// TwinCAT 3 PLC project PLC_HMI_ACCT_1
// ProgramVersion: 3.1.4026.19
// libraries:
//   Tc2_DataExchange, * (Beckhoff Automation GmbH)
//   Tc2_IoFunctions, * (Beckhoff Automation GmbH)
//   Tc2_MC2, * (Beckhoff Automation GmbH)
//   Tc2_Standard, * (Beckhoff Automation GmbH)
//   Tc2_System, * (Beckhoff Automation GmbH)
//   Tc2_Utilities, * (Beckhoff Automation GmbH)
//   Tc3_Database, * (Beckhoff Automation GmbH)
//   Tc3_EventLogger, * (Beckhoff Automation GmbH)
//   Tc3_Module, * (Beckhoff Automation GmbH)
// project tree:
//   DUTs/ ST_Alarm.TcDUT, ST_Error_Station_Handling.TcDUT, ST_Error_Description_Handling.TcDUT, ST_For_Screen.TcDUT, ST_For_Screen_New.TcDUT, ST_Recipe_Changes.TcDUT, ST_UserManagment.TcDUT, S_Information.TcDUT, S_Information_Text.TcDUT, S_LogData.TcDUT
//   FB/ FB_GetSystemTime.TcPOU, FB_Persistent.TcPOU, FB_ReadWriteLogCSV.TcPOU, FB_Save.TcPOU, FB_SaveLineToFile.TcPOU, FB_SaveTextToFile.TcPOU
//   FB/RecipeCSV/ FB_ListSaveCSV.TcPOU, FB_LoadCSV.TcPOU, FB_RecipeSaveCSV.TcPOU, FB_RecipeVariablesSaveCSV.TcPOU
//   FB/RecipeList/ E_FileOpSteps.TcDUT, FB_Load.TcPOU
//   GVLs/ GVL_CFG.TcGVL, GVL_Error.TcGVL, GVL_Gauge.TcGVL, GVL_Recipe.TcGVL, GVL_Screw.TcGVL, GVL_USER.TcGVL
//   NotUsedPOU/ P_50_screw.TcPOU, P_Error_Handling.TcPOU
//   / PlcTask.TcTTO
//   POUs/ADS/ P_ADS_Gauge.TcPOU, P_ADS_OEE.TcPOU, P_ADS_Screw.TcPOU
//   POUs/DataLogging/ p_24h_C1_2.TcPOU, p_24h_C2_2.TcPOU, P_ArrayToFile.TcPOU, P_CameraFlip.TcPOU, P_Gauge_Measures.TcPOU, P_OEE_Raport.TcPOU, P_Recipebackup.TcPOU, P_RecipeChange.TcPOU, P_ScrewersCharts_1.TcPOU, P_ScrewersCharts_2.TcPOU
//   POUs/ MAIN.TcPOU, P_Time.TcPOU
//   POUs/Persistent/ P_Persistent.TcPOU, P_PersistentDataSave.TcPOU
//   POUs/Users/ P_UserManagment.TcPOU
// (motion and I/O tree: see PLC project programplc)
// real-time tasks:
//   TASK MainTask: cycle T#3ms, priority 20, ADS port 350
//   TASK SafetyTask: cycle T#10ms, priority 22, ADS port 351
//   TASK WeightTask: cycle T#2ms, priority 19, ADS port 354
//   TASK PlcTask: cycle T#10ms, priority 21, ADS port 355
//   TASK TaskToRefreshEAP: cycle T#1ms, priority 12, ADS port 301
// variable links:

CONFIGURATION PLC_HMI_ACCT_1
    RESOURCE PLC ON TwinCAT3
        TASK PlcTask(INTERVAL := T#10ms, PRIORITY := 21);
        PROGRAM MAIN WITH PlcTask : MAIN;
    END_RESOURCE
END_CONFIGURATION

// ---- DUTs/ST_Alarm.TcDUT
TYPE ST_Alarm :
STRUCT
	sTekst1				: WSTRING(255);
	sTekst2				: WSTRING(255);
	sTekst3				: WSTRING(255);
	dtUtworzenia		: DT;
	iNumer				: INT;
	historical_alarm	: WSTRING(1000);
END_STRUCT
END_TYPE

// ---- DUTs/ST_Error_Station_Handling.TcDUT
TYPE ST_Error_Station_Handling :
STRUCT
	udiStationInError			:UDINT;
	wsStasionInError				:WSTRING(255);
END_STRUCT
END_TYPE

// ---- DUTs/ST_Error_Description_Handling.TcDUT
TYPE ST_Error_Description_Handling :
STRUCT
	udiStationErrorCode		:UDINT;
	wsStationErrorDescription	:WSTRING(255);	
END_STRUCT
END_TYPE

// ---- DUTs/ST_For_Screen.TcDUT
TYPE ST_For_Screen :
STRUCT
	data				:WSTRING(255);
	alarmy				:WSTRING(1000);
	user				:WSTRING(80);
	bErrorOccure		:BOOL := FALSE;
END_STRUCT
END_TYPE

// ---- DUTs/ST_For_Screen_New.TcDUT
TYPE ST_For_Screen_New :
STRUCT
	data				:WSTRING(255);
	alarmy				:WSTRING(1000);
	alarmy_id			:UDINT;
	stacja				:UDINT;
	user				:WSTRING(80);
	bErrorOccure		:BOOL := FALSE;
END_STRUCT
END_TYPE

// ---- DUTs/ST_Recipe_Changes.TcDUT
TYPE ST_Recipe_Changes :
STRUCT
	old_value :LREAL;
	new_value :LREAL;
	who_changed :WSTRING(200);
	when_changed :DT;	
	which_param_name :WSTRING(200);
	which_param_var	 :WSTRING(200);	
	which_param_cntr :WSTRING(200);
	which_recipe :WSTRING(200);
	
END_STRUCT
END_TYPE

// ---- DUTs/ST_UserManagment.TcDUT
TYPE ST_UserManagment :
STRUCT
	userID 				:	INT;			//numer porządkowy użytkownika
//	domain				:	STRING(80);
	enabled				:	BOOL;
	userLogin			:	STRING(80);		//login do zalogowania
	userNameSurname 	:	WSTRING(255);	//imię i nazwisko
	userNameSurnameNumber	:UINT;
	password			:	STRING(255);	//hasło kalwiaturowe
	passwordRFID		:	STRING(255);	//hasło rfid
	passwordQR			:	STRING(255);	//hasło qr
	userGroup			:	STRING(80);		//grupa użytkowników
	userGropuNumber		:	UINT;			//numer grupy
//	autoLogOff			:	STRING(80);		//czas do wylogowania
//	locale				:	STRING(80);		//gdzie zapisujemy
//	timeFormatlocale	:	STRING(80);		//format godziny
//	timeZone			:	STRING(80);		//strefa czasowa
	signedPassword		:	STRING(80);		//hasło przekazywane do HMI
END_STRUCT
END_TYPE

// ---- DUTs/S_Information.TcDUT
(*
Nazwa:			S_Error
Opis:			Struktura bledu
Wersja:			v0.2
Data:			2018-10-10
Autor:			TW
Urzadzenia:		
Konfiguracja:	
Info:
- dodano string2
*)
TYPE S_Information :
STRUCT 
	udiID				: UDINT;
	wsDescription		: WSTRING;
END_STRUCT
END_TYPE

// ---- DUTs/S_Information_Text.TcDUT
(*
Nazwa:			S_Error
Opis:			Struktura bledu
Wersja:			v0.2
Data:			2018-10-10
Autor:			TW
Urzadzenia:		
Konfiguracja:	
Info:
- dodano string2
*)
TYPE S_Information_Text :
STRUCT 
	desc				: WSTRING;
	wsDescription		: WSTRING;
END_STRUCT
END_TYPE

// ---- DUTs/S_LogData.TcDUT
TYPE S_LogData :
STRUCT
END_STRUCT
END_TYPE

// ---- FB/RecipeList/E_FileOpSteps.TcDUT
{attribute 'qualified_only'}
{attribute 'strict'}
TYPE E_FileOpSteps :
(
	eNop 					:=	0,
	eStartOpen				:=	10,
	eWaitOpen				:=	20,
	eStartOper				:=	30,
	eWaitOper				:=	40,
	eStartClose				:=	50,
	eWaitClose				:=	60
);
END_TYPE

// ---- GVLs/GVL_CFG.TcGVL
{attribute 'qualified_only'}
VAR_GLOBAL PERSISTENT
	//butelki
	bBottleBuPu :BOOL:=FALSE;
	bBottlePI :BOOL:=TRUE;
	bBottleUBF :BOOL:=TRUE;
	bNoBottleFeed	:BOOL:=FALSE;
	
	//nasadki
	bCapUCF :BOOL:=TRUE;
	bCapSO :BOOL:=FALSE;
	bCapWibro :BOOL:=FALSE;
	bCapGiraffe :BOOL:=FALSE;
	bNoCapFeed	:BOOL:=FALSE;
	
	//maszyna
	bPlatinsCFG :BOOL:=TRUE;
	bTwoPhaseCFG :BOOL:=TRUE;;
	bAirless :BOOL:=FALSE;
	bROPP :BOOL:=FALSE;;
	
	sIP	:STRING:='192.168.40.180.1.1';
	sPort :T_AmsPort:=851;
	
	sRightTime	:STRING;
	tbreakTime_1:STRING:='10:35:00';
	tbreakTime_2:STRING:='14:35:00';
	bBreakReset:BOOL;
	
	bWenglorCapPutted :BOOL;
	bWenglorCapCorrect :BOOL;
	
END_VAR

// ---- GVLs/GVL_Error.TcGVL
{attribute 'qualified_only'}
(**VAR_GLOBAL PERSISTENT
	udi_Station_In_Error			:UDINT;
	udi_Station_In_Error_Code		:UDINT;
	ws_Stasion_In_Error				:WSTRING;
	ws_Station_Error_Description		:WSTRING(255);
	ws_Station_Error_Description_2	:WSTRING(255);
	A_Error_station	:ARRAY[0..100] OF ST_Error_Station_Handling; 
	A_Error_description	:ARRAY[0..500] OF ST_Error_Description_Handling;
	
	b_empy_error					:BOOL;
	b_new_system					:BOOL;
	
	sVisGuid						:STRING;
	
	b_reset_event_logger :BOOL;
END_VAR**)
VAR_GLOBAL
	b_reset_event_logger :BOOL;
	logowanie_krok: INT;
	b_cameras_ivms:BOOL;
END_VAR

// ---- GVLs/GVL_Gauge.TcGVL
{attribute 'qualified_only'}
VAR_GLOBAL
	//input
	lr_WeightMass_recipe	:LREAL;
	lr_Dispencer1WeightMeasured	:LREAL;
	lr_Dispencer2WeightMeasured	:LREAL;
	lr_Dispencer3WeightMeasured	:LREAL;
	lr_Dispencer4WeightMeasured	:LREAL;
	lr_Tolerance_Low			:LREAL;
	lr_Tolerance_High			:LREAL;
	lr_weight_measured_1		:LREAL;
	lr_weight_measured_2		:LREAL;
	lr_weight_measured_3		:LREAL;
	lr_weight_measured_4		:LREAL;
	
	lr_mass_value_1				:LREAL;
	lr_mass_value_2				:LREAL;
	lr_mass_value_3				:LREAL;
	lr_mass_value_4				:LREAL;
	
	
	//output
	lr_out_max_weight_value :LREAL;
	lr_out_min_tolerance_low :LREAL;
	lr_out_max_tolerance_high :LREAL;
	
	lr_out_weight_measured_1 :LREAL;
	lr_out_weight_measured_2 :LREAL;
	lr_out_weight_measured_3 :LREAL;
	lr_out_weight_measured_4 :LREAL;
	
	s_actual_weight_1	:STRING;
	s_actual_weight_2	:STRING;	
	s_actual_weight_3	:STRING;
	s_actual_weight_4	:STRING;
	
	s_actual_weight_1_diff	:STRING;
	s_actual_weight_2_diff	:STRING;
	s_actual_weight_3_diff	:STRING;
	s_actual_weight_4_diff	:STRING;

	s_actual_corr_1		:STRING;
	s_actual_corr_2		:STRING;
	s_actual_corr_3		:STRING;
	s_actual_corr_4		:STRING;	
	
	s_actual_dose_1		:STRING;
	s_actual_dose_2		:STRING;
	s_actual_dose_3		:STRING;
	s_actual_dose_4		:STRING;
	
	lr_corr_add_1	:LREAL;
	lr_corr_sub_1	:LREAL;
	lr_corr_add_2	:LREAL;
	lr_corr_sub_2	:LREAL;
	lr_corr_add_3	:LREAL;
	lr_corr_sub_3	:LREAL;
	lr_corr_add_4	:LREAL;
	lr_corr_sub_4	:LREAL;
	
	s_actual_torque_1	:STRING;
	s_actual_torque_2	:STRING;
	s_actual_torque_diff_1		:STRING;
	s_actual_torque_diff_2		:STRING;
	
	s_actual_level_1	:STRING;
	s_actual_level_2	:STRING;
	
	lr_out_torque_low_1		:LREAL;
	lr_out_torque_low_2		:LREAL;
	lr_out_torque_high_1		:LREAL;
	lr_out_torque_high_2		:LREAL;	
	
	s_out_weight_measured_1 :STRING;
	s_out_weight_measured_2 :STRING;
	s_out_weight_measured_3 :STRING;
	s_out_weight_measured_4 :STRING;

	lr_diff_dispencer_1:LREAL;
	lr_diff_dispencer_2:LREAL;
	
	s_time_mainscreen:WSTRING(80);
	
	bDosingTwoPhasesShow	:BOOL;
END_VAR

// ---- GVLs/GVL_Recipe.TcGVL
{attribute 'qualified_only'}
VAR_GLOBAL PERSISTENT
	b_recipe_backup	:BOOL;
	
	b_recipe_bool_change :BOOL; //sygnał, że ktoś zmienił parametr bool
	b_recipe_real_change :BOOL; //sygnał, że ktoś zmienił parametr inny
	i_recipe_change :INT;
	lr_recipe_change :LREAL; //stara wartość w polu lr_param
	
	b_recipe_change_1 :BOOL;
	i_recipe_change_1 :INT;
	lr_recipe_change_1 :LREAL; //nowa wartość w polu lr_param
	
	s_recipe_change    :WSTRING(200); //kto zmienił parametr
	s_recipe_change_1  :WSTRING(200); //jaki parametr
	s_recipe_change_2  :WSTRING(200); //zmienna receptury
	s_recipe_change_3  :WSTRING(300); //zmienna do kontrolki
	b_old_recipe_param :BOOL; //stara wartość parametru b_param
	b_new_recipe_param :BOOL; //nowa wartość parametru b_param
	

	
	s_recipe_value :STRING;
	ArRecipeChanges: ARRAY [0..500] OF st_recipe_changes;	
	s_recipe_name :WSTRING(200); //nazwa receptury
	s_recupe_change_4 :WSTRING(200);
	b_recipe_changes_clear :BOOL:=FALSE;
END_VAR

// ---- GVLs/GVL_Screw.TcGVL
{attribute 'qualified_only'}
VAR_GLOBAL
	 aLast50Screw1: ARRAY[1..501] OF LREAL;
	 aLast50Screw2: ARRAY[1..501] OF LREAL;
	 bExport:BOOL;
	 a50ScrewSetted1: ARRAY[1..501] OF LREAL;
	 a50ScrewSetted2: ARRAY[1..501] OF LREAL;
END_VAR

// ---- GVLs/GVL_USER.TcGVL
{attribute 'qualified_only'}
VAR_GLOBAL PERSISTENT
	user_array 					: ARRAY[1..100] OF ST_UserManagment;  // Tablica użytkowników
    currentUser 				: INT := 1;  // Indeks bieżącego użytkownika (zaczyna od 1)
	outside_login_pool			:STRING(255);  
	currentUserName 			:WSTRING(255);
	currentUserGroup			:STRING(80);
	currentUserGroupNumber		:UINT;
	putted_user_password		:STRING(255);  //pole w które użytkownik wpisuje hasło
	newuserNameSurname 			:WSTRING(255);	//imię i nazwisko
	newpassword					:STRING(255);	//hasło
	newpasswordRFID				:STRING(255);	//hasło rfid
	newpasswordQR				:STRING(255);	//hasło qr
	newuserGroup				:STRING(80);		//grupa użytkowników
	newuserGroupNumber			:UINT;
	newautoLogOff				:STRING(80);			//czas do wylogowania
	actual_editted_user			:WSTRING(255);	//wybór aktualnie edytowanego użytkownika
	edituserNameSurname 		:WSTRING(255);	//imię i nazwisko
	editpassword				:STRING(255);	//hasło
	editpasswordRFID			:STRING(255);	//hasło rfid
	editpasswordQR				:STRING(255);	//hasło qr
	edituserGroup				:STRING(80);	//grupa użytkowników
	editUserGroupNumber			:UINT;
	editautoLogOff				:STRING(80);	//czas do wylogowania


END_VAR
VAR_GLOBAL
	new_user_add_error			:BOOL;
	edit_user_error				:BOOL;
	bwait						:BOOL;
	delete_user					:BOOL;
	delete_user_accept			:BOOL;
	delete_user_error			:BOOL;
	choosen_to_delete			:WSTRING(255);
	user_deleted_succes			:BOOL;
	password_to_log_in			:STRING(80); //hasło do pola (1 z 5 (adm, opr, ser, tech, mech	
	b_rewrite_users_after_issues:BOOL:=FALSE;
	b_user_drop_the_login		:BOOL;
	i_choosen_language 			:INT:=1;
	outside_accept_login		:BOOL;
	logout						:BOOL;
	user_try_to_log				:BOOL;
	user_accept_to_log_in		:BOOL;
	no_user_found				:BOOL;
	user_succesed_log			:BOOL;
	edit_user_qr_or_rfid_password :BOOL;		//edycja kodów rfid lub qr
	new_user_added				:BOOL;		//dodano użytkownika w PLC
	user_eddited				:BOOL; 		//zedytowano użytkownika w PLC
	b_new_users					:BOOL;		//wgranie uzytkowników
	new_user					:BOOL;			//inicjalizacja dodawania nowego użytkownika
	new_user_accept				:BOOL;			//akceptacja dodania nowego użytkownika
	edit_user					:BOOL;				//inicjalizacja edycji użytkownika
	edit_user_accept			:BOOL;			//akceptacja edycji użytkownika
	actualUserOn_UserName		:STRING(80);
	b_rewrite_main_users		:BOOL:=FALSE;
	string_of_properties 		: STRING(1000);  // String z HMI z danymi użytkowników
END_VAR

// ---- POUs/MAIN.TcPOU
PROGRAM MAIN
VAR
		
END_VAR

//P_ADS_1();
P_Time();
//P_History_New();
P_UserManagment();
P_Recipebackup();
P_Gauge_Measures();
P_ADS_Gauge();
//P_ADS_Err();
//P_Error_Handling();
P_RecipeChange();
P_ArrayToFile();
P_ScrewersCharts_1();
P_ScrewersCharts_2();
P_ADS_Screw();
P_24h_C1_2();
P_24h_C2_2();
//P_HistoryWarning();
P_CameraFlip();
//P_EventLogger();
//P030_Recipes();
//P010_AlarmsWarningsInfosLogs();
//P020_RtcEffectivityOEE();
//P009_ReadSavePersistent();
P_OEE_Raport();
P_ADS_OEE();
P_PersistentDataSave();
P_Persistent();

END_PROGRAM

// ---- POUs/P_Time.TcPOU
PROGRAM P_Time
VAR
    fbSystemTime : GETSYSTEMTIME;
	fbSystemTime2 : FB_GetSystemTime;
    timeAsFileTime : T_FILETIME;
    timeAsDT : DT;
	actual_date_meawhile :DT;
	s_time_mainscreen	:WSTRING(80);
	tonBreakTurnOff 	:TON;
END_VAR

tonBreakTurnOff(IN:=gvl_cfg.bBreakReset,PT:=T#5S);
fbSystemTime2(bEnable:=TRUE);
fbSystemTime(
    timeLoDW => timeAsFileTime.dwLowDateTime,
    timeHiDW => timeAsFileTime.dwHighDateTime 
);
(*timeAsDT := FILETIME_TO_DT(timeAsFileTime);
actual_date_meawhile:=timeAsDT;
actual_date_meawhile := actual_date_meawhile + T#2H;
s_time_mainscreen := DT_TO_WSTRING(actual_date_meawhile);
s_time_mainscreen := WRIGHT(s_time_mainscreen, WLEN(s_time_mainscreen) - 3);
gvl_his.s_time_mainscreen:=s_time_mainscreen;
gvl_cfg.wsRightTime:=WRIGHT(s_time_mainscreen,8);*)
timeAsDT :=fbSystemTime2.dtActTime;
actual_date_meawhile:=timeAsDT;
s_time_mainscreen := DT_TO_WSTRING(actual_date_meawhile);
s_time_mainscreen := WRIGHT(s_time_mainscreen, WLEN(s_time_mainscreen) - 3 );
gvl_gauge.s_time_mainscreen:=s_time_mainscreen;


IF gvl_cfg.sRightTime = gvl_cfg.tbreakTime_1 OR gvl_cfg.sRightTime = gvl_cfg.tbreakTime_2 THEN
	gvl_cfg.bBreakReset:=TRUE;
END_IF

IF tonBreakTurnOff.Q THEN
	gvl_cfg.bBreakReset:=FALSE;
END_IF

END_PROGRAM

// ---- FB/FB_GetSystemTime.TcPOU
(****************************************************************************************)
(*							Beckhoff Automation Poland									*)
(*								FB_GetSystemTime  v1.2									*)
(*									26.07.2013											*)
(*		v1.2 - zmiana nazwy bloku z FB_Time na FB_GetSystemTime, dodanie wyjscia DT		*)
(*		v1.1 - dodano na wyjściu zmienną czasu w formie struktury TIMESTRUCT 			*)
(*				Blok funkcyjny podający dokładną datę w odrębnych zmiennych				*)
(*						może być wywołany raz w programie PLC							*)
(*						Wymaga dodania biblioteki TcUtilities.lib						*)
(*______________________________________________________________________________________*)
FUNCTION_BLOCK FB_GetSystemTime
VAR_INPUT
	bEnable:			BOOL;				(*Aktywuje pobieranie czasu systemowego*)
END_VAR
VAR_OUTPUT
	stActTime			:	TIMESTRUCT;
	dtActTime: DT;
(*Poszczególne składowe daty*)
	wYear 				:	WORD;
	wMonth 				:	WORD;
	wDayOfWeek 			: 	WORD;
	wDay 				:	WORD;
	wHour 				:	WORD;
	wMinute 			:	WORD;
	wSecond 			:	WORD;
	wMilliseconds 		: 	WORD;
END_VAR
VAR
	fbGetTime			:	NT_GetTime;
	Get					:	TON;
END_VAR
VAR CONSTANT
	tFrequency			:	TIME			:= T#1s;				(*Częstotliwość pobierania czasu*)
END_VAR

Get(IN:= NOT Get.Q AND bEnable, PT:=tFrequency);
fbGetTime(
	NETID:= '',
	START:= Get.Q,
	TMOUT:= T#200ms,
	TIMESTR=>stActTime);

dtActTime 		:= SYSTEMTIME_TO_DT(stActTime);
wDay 			:= stActTime.wDay;
wDayOfWeek 		:= stActTime.wDayOfWeek;
wHour 			:= stActTime.wHour;
wMilliseconds 	:= stActTime.wMilliseconds;
wMinute 		:= stActTime.wMinute;
wMonth 			:= stActTime.wMonth;
wSecond 		:= stActTime.wSecond;
wYear 			:= stActTime.wYear;

END_FUNCTION_BLOCK

// ---- POUs/Users/P_UserManagment.TcPOU
PROGRAM P_UserManagment
VAR	
	user_log				:BOOL 				:= GVL_USER.user_try_to_log;           	//użytkownik wywołał okno logowania
	user_accept				:BOOL 				:= GVL_USER.user_accept_to_log_in;     	//użytkownik zaakceptował hasło
	outside_login_accept	:BOOL				:= gvl_user.outside_accept_login;		//przekazanie potwierdzenia procesu logowania
	user_login_error		:BOOL 				:= GVL_USER.no_user_found;				//brak dopasowanego użytkownika
	user_log_succes			:BOOL 				:= GVL_USER.user_succesed_log;			//zalogowano z powodzeniem
	i,j,z					:INT;														//zmienne dla warunków
	bprzypisanie			:BOOL;
	btest					:BOOL:=FALSE;
	k						:INT;
	userExists				:BOOL;														//zmienne dla programu
	outside_login_pool		:STRING(255)		:= gvl_user.outside_login_pool;												//przekazanie loginu do wizualizacji
	user_password			:STRING(255) 		:= GVL_USER.putted_user_password;		//wprowadzone użytkownikiem hasło
	b_new_users				:BOOL;									
	delayTimer: TON;  // Timer do opóźnienia o 500 ms					//nowe wgranie użytkowników
	allowedGroups : ARRAY[1..5] OF STRING(80) := ['Admin', 'Mechanik', 'Operator', 'Technolog', 'Serwis'];
	allowedGroupsNumber	:ARRAY[1..5] OF UINT:=[1,2,3,4,5];
	validGroup    : BOOL;  // Zmienna do walidacji grupy
    uniqueUser    : BOOL;  // Zmienna sprawdzająca unikalność hasła
    freeSlot      : BOOL;  // Zmienna wskazująca wolne miejsce na nowego użytkownika
	bwait	:BOOL :=gvl_user.bwait; //ekran oczekiwania na plc
	bClear	:BOOL:=FALSE;
	iClearArrayNr :INT;
	
	actual_user : WSTRING(255);
	

	new_user				:BOOL := GVL_USER.new_user;			//inicjalizacja dodania nowego użytkownika
	new_user_accept			:BOOL := GVL_USER.new_user_accept;			//akceptacja dodania użytkownika z ekranu
	new_user_added			:BOOL := GVL_USER.new_user_added;			//udane dodanie użytkownika
	new_user_add_error		:BOOL := GVL_USER.new_user_add_error;			//nieudane dodawanie
	newautoLogOff			:STRING(80) := GVL_USER.newautoLogOff;			//czas do wylogowania
	newuserNameSurname 		:WSTRING(255)  := GVL_USER.newuserNameSurname;	//imię i nazwisko				
	newpassword				:STRING(255) := GVL_USER.newpassword;	//hasło
	newpasswordRFID			:STRING(255) := GVL_USER.newpasswordRFID;	//hasło rfid
	newpasswordQR			:STRING(255) := GVL_USER.newpasswordQR;	//hasło qr
	newuserGroup			:STRING(80) := GVL_USER.newuserGroup;		//grupa użytkowników
	newuserLogoffbetween 	:STRING(80);
	
	edit_user						:BOOL := GVL_USER.edit_user;	//inicjalizacja edycji parametrów użytkownika
	edit_user_accept				:BOOL := GVL_USER.edit_user_accept;	//akceptacja wprowadzonych zmiennych z ekranu
	user_eddited					:BOOL := GVL_USER.user_eddited;	//odpowiedź z plc do hmi - udana edycja
	edit_user_qr_or_rfid_password	:BOOL := GVL_USER.edit_user_qr_or_rfid_password;	//edycja rfid lub qr dopisanego do użytkownika
	edit_user_error					:BOOL := GVL_USER.edit_user_error;			//odpowiedź z plc do hmi - nieudana edycja uzytkownika
	editautoLogOff					:STRING(80) := GVL_USER.editautoLogOff;			//czas do wylogowania użytkownika
	edituserNameSurname 			:WSTRING(255) := GVL_USER.edituserNameSurname ;	//imię i nazwisko
	editpassword					:STRING(255) := GVL_USER.editpassword;	//hasło
	editpasswordRFID				:STRING(255) := GVL_USER.editpasswordRFID;	//hasło rfid
	editpasswordQR					:STRING(255) := GVL_USER.editpasswordQR;	//hasło qr
	edituserGroup					:STRING(80) := GVL_USER.edituserGroup;	//grupa użytkowników
	edituserLogoffbetween 	:STRING(80);

	userExists_2			:BOOL;
	userExists_3			:BOOL;
	
	bFirstCycle				:BOOL := FALSE;
	
	iValueForCheck			:INT;
	logowanie_krok	:INT;
	bLogOffUserReset :BOOL;
	tonLogOffUser :ton;
END_VAR


bFirstCycle:=TRUE; //Symulacja 1 cyklu sterownika
tonLogOffUser(IN:=(NOT (GVL_USER.currentUserName="Niezalogowany Użytkownik")) AND (NOT bLogOffUserReset) AND (NOT (GVL_USER.currentUserName="Operator")), PT:=T#60M);


IF bClear THEN 
    // Sprawdzamy, czy numer wiersza mieści się w zakresie tablicy
    IF (iClearArrayNr >= 1) AND (iClearArrayNr <= 100) THEN
        // Czyszczenie wybranego wiersza tablicy
        GVL_USER.user_array[iClearArrayNr].userID := 0;
        //GVL_USER.user_array[iClearArrayNr].domain := '';
        GVL_USER.user_array[iClearArrayNr].enabled := FALSE;
        GVL_USER.user_array[iClearArrayNr].userLogin := '';
        GVL_USER.user_array[iClearArrayNr].userNameSurname := "";  // WSTRING wymaga również pustego ciągu znaków
        GVL_USER.user_array[iClearArrayNr].password := '';
        GVL_USER.user_array[iClearArrayNr].passwordRFID := 'tup';
        GVL_USER.user_array[iClearArrayNr].passwordQR := 'tup';
        GVL_USER.user_array[iClearArrayNr].userGroup := '';
       // GVL_USER.user_array[iClearArrayNr].autoLogOff := '';
        //GVL_USER.user_array[iClearArrayNr].locale := '';
        //GVL_USER.user_array[iClearArrayNr].timeFormatlocale := '';
        //GVL_USER.user_array[iClearArrayNr].timeZone := '';
        GVL_USER.user_array[iClearArrayNr].signedPassword := '';
    END_IF

    // Resetowanie flagi bClear po wykonaniu czyszczenia
    bClear := FALSE;
END_IF

// Proces logowania użytkownika GVL_USER.user_try_to_log AND
IF  GVL_USER.user_accept_to_log_in THEN
    GVL_USER.user_succesed_log := FALSE;
    GVL_USER.no_user_found := TRUE;
    gvl_user.bwait := TRUE;
	iValueForCheck:=1;    
	userExists_3 := FALSE;	
    FOR i := 1 TO 100 DO
		
        IF GVL_USER.user_array[i].password = GVL_USER.putted_user_password OR 
           (GVL_USER.user_array[i].passwordRFID = GVL_USER.putted_user_password) OR 
           (GVL_USER.user_array[i].passwordQR = GVL_USER.putted_user_password) THEN
		   
            GVL_USER.currentUser := i;
            userExists_3 := TRUE;
			iValueForCheck:=2;
            EXIT;
			
        END_IF
		
    END_FOR

    IF NOT userExists_3 THEN
		
        GVL_USER.no_user_found := TRUE;
        gvl_user.bwait := FALSE;
		userExists_3 := FALSE;
		iValueForCheck:=3;
		GVL_USER.currentUser := 6;
		gvl_user.currentUserName :="Niezalogowany Użytkownik";
		gvl_user.currentUserGroup :='Niezalogowany';
		gvl_user.currentUserGroupNumber :=0; //
        GVL_USER.user_succesed_log := TRUE;  // Potwierdzenie, że wylogowanie i logowanie zakończyły się sukcesem
        GVL_USER.logout := FALSE;  // Resetowanie sygnału wylogowania
		GVL_USER.putted_user_password:='';
    ELSE

        FOR i := 1 TO 100 DO
            // Sprawdzenie, czy użytkownik jest aktywny
            IF GVL_USER.user_array[i].enabled THEN
                // Sprawdzenie, czy wprowadzone hasło odpowiada loginowi lub RFID/QR
                GVL_USER.no_user_found := FALSE;
				iValueForCheck:=4;
                IF (GVL_USER.user_array[i].password = GVL_USER.putted_user_password) OR
                   (GVL_USER.user_array[i].passwordRFID = GVL_USER.putted_user_password) OR
                   (GVL_USER.user_array[i].passwordQR = GVL_USER.putted_user_password) THEN
                   //delayTimer(IN := TRUE, PT := T#1S);
				   iValueForCheck:=5;
                    // Jeśli wprowadzony kod to RFID lub QR, zastąp go przypisanym hasłem
                    IF GVL_USER.user_array[i].passwordRFID = GVL_USER.putted_user_password THEN
                        GVL_USER.putted_user_password := GVL_USER.user_array[i].password;
						iValueForCheck:=6;
                    	ELSIF GVL_USER.user_array[i].passwordQR = GVL_USER.putted_user_password THEN
                        	GVL_USER.putted_user_password := GVL_USER.user_array[i].password;
							iValueForCheck:=6;
                    END_IF

                 // Sprawdzanie grupy użytkownika i przypisanie odpowiedniej wartości
                 	IF GVL_USER.user_array[i].userGroup = 'Admin' THEN
						iValueForCheck:=7;
                        gvl_user.password_to_log_in := GVL_USER.user_array[i].signedPassword;
                    	ELSIF GVL_USER.user_array[i].userGroup = 'Operator' THEN
                        	gvl_user.password_to_log_in := GVL_USER.user_array[i].signedPassword;
                    	ELSIF GVL_USER.user_array[i].userGroup = 'Serwis' THEN
                        	gvl_user.password_to_log_in := GVL_USER.user_array[i].signedPassword;
                    	ELSIF GVL_USER.user_array[i].userGroup = 'Technolog' THEN
                       		gvl_user.password_to_log_in := GVL_USER.user_array[i].signedPassword;
                    	ELSIF GVL_USER.user_array[i].userGroup = 'Mechanik' THEN
                        	gvl_user.password_to_log_in := GVL_USER.user_array[i].signedPassword;
                    END_IF
                    //IF delayTimer.Q THEN
                		//delayTimer(IN := FALSE);
						iValueForCheck:=8;
						gvl_user.currentUserName := GVL_USER.user_array[i].userNameSurname;
						gvl_user.currentUserGroup := GVL_USER.user_array[i].userGroup;
						gvl_user.currentUserGroupNumber := GVL_USER.user_array[i].userGropuNumber;
                    	GVL_USER.user_succesed_log := TRUE;
                    	GVL_USER.no_user_found := FALSE;                   
                    	gvl_user.bwait := FALSE;
                    	GVL_USER.user_try_to_log := FALSE;
                    	GVL_USER.user_accept_to_log_in := FALSE;
                    // Zerowanie zmiennych po udanym logowaniu
					//gvl_user.outside_accept_login := TRUE;  // Informacja dla wizualizacji
                    //GVL_USER.putted_user_password := '';   // Wyczyszczenie wprowadzonego hasła
                    // Wyczyszczenie hasła do logowania
					//gvl_user.password_to_log_in := '';
					//userExists_3 := FALSE;
					END_IF					
                END_IF
            
        END_FOR
		
        // Jeżeli pętla się zakończy i nie znaleziono użytkownika
        IF NOT GVL_USER.user_succesed_log THEN
            GVL_USER.no_user_found := TRUE; // Ustaw błąd logowania
            gvl_user.bwait := FALSE;
			userExists_3 := FALSE;
			GVL_USER.user_succesed_log := FALSE;
			GVL_USER.putted_user_password:='';
			iValueForCheck:=9;
        END_IF
    END_IF
	GVL_USER.user_succesed_log := FALSE;
	userExists_3:=FALSE;
END_IF


// Dodawanie nowego użytkownika
IF GVL_USER.new_user AND GVL_USER.new_user_accept THEN
    GVL_USER.new_user_added := FALSE;
    GVL_USER.new_user_add_error := TRUE;
	gvl_user.bwait := TRUE;
    validGroup := FALSE;  // Na początku zakładamy, że grupa nie jest poprawna
    uniqueUser := TRUE;   // Na początku zakładamy, że hasło jest unikalne
    freeSlot := FALSE;    // Na początku zakładamy, że nie ma wolnego miejsca
    
    // Sprawdzanie, czy wybrana grupa jest jedną z dozwolonych GVL_USER.newuserGroup = allowedGroups[j] 
    FOR j := 1 TO 5 DO
        IF GVL_USER.newuserGroupNumber = allowedGroupsNumber[j]	THEN
            	validGroup := TRUE;  // Jeśli grupa jest dozwolona, ustawiamy na TRUE
        END_IF
    END_FOR

    // Jeśli grupa nie jest poprawna, przerywamy proces dodawania użytkownika
    IF NOT validGroup THEN
        GVL_USER.new_user_add_error := TRUE;
    ELSE
        // Sprawdzanie, czy hasło nie jest już przypisane do innego użytkownika
        FOR i := 7 TO 100 DO
            IF GVL_USER.user_array[i].enabled AND 
               ((GVL_USER.user_array[i].password = GVL_USER.newpassword) OR 
                (GVL_USER.user_array[i].passwordRFID = GVL_USER.newpasswordRFID) OR 
                (GVL_USER.user_array[i].passwordQR = GVL_USER.newpasswordQR)) THEN
                uniqueUser := FALSE;  // Jeśli hasło, RFID lub QR istnieje, ustawiamy na FALSE
            END_IF
        END_FOR

        // Jeśli hasło jest unikalne, szukamy wolnego miejsca w tablicy
        IF uniqueUser THEN
            FOR i := 10 TO 100 DO
                IF NOT GVL_USER.user_array[i].enabled THEN
                    // Przypisanie danych nowego użytkownika
                    GVL_USER.user_array[i].userID := i;
                    GVL_USER.user_array[i].userLogin := GVL_USER.newpassword; // Używamy loginu z hasła
                    GVL_USER.user_array[i].userNameSurname := GVL_USER.newuserNameSurname;
                    GVL_USER.user_array[i].password := GVL_USER.newpassword;

                    // Sprawdzanie, czy pole RFID jest puste - jeśli tak, zapisujemy "tup"
                    IF GVL_USER.newpasswordRFID = '' THEN
                        GVL_USER.user_array[i].passwordRFID := 'tup';
                    ELSE
                        GVL_USER.user_array[i].passwordRFID := GVL_USER.newpasswordRFID;
                    END_IF

                    // Sprawdzanie, czy pole QR jest puste - jeśli tak, zapisujemy "tup"
                    IF GVL_USER.newpasswordQR = '' THEN
                        GVL_USER.user_array[i].passwordQR := 'tup';
                    ELSE
                        GVL_USER.user_array[i].passwordQR := GVL_USER.newpasswordQR;
                    END_IF
                    newuserLogoffbetween:= CONCAT('PT',GVL_USER.newautoLogOff);
                    GVL_USER.user_array[i].userGroup := GVL_USER.newuserGroup;  // Grupa musi być poprawna
                    //GVL_USER.user_array[i].autoLogOff := Concat(newuserLogoffbetween,'M');
                    GVL_USER.user_array[i].enabled := TRUE;
					//gvl_user.user_array[i].locale:='client';
					//gvl_user.user_array[i].timeFormatlocale:='project';
					//gvl_user.user_array[i].timeZone:='project';
					//gvl_user.user_array[i].domain:='TcHmiUserManagment';
					
					IF GVL_USER.newuserGroupNumber =1 THEN
                        GVL_USER.user_array[i].signedPassword := 'adm';
						GVL_USER.user_array[i].userGropuNumber :=1;
                    ELSIF GVL_USER.newuserGroupNumber =3 THEN
                        GVL_USER.user_array[i].signedPassword := 'opr';
						GVL_USER.user_array[i].userGropuNumber :=3;
                    ELSIF GVL_USER.newuserGroupNumber =5 THEN
                        GVL_USER.user_array[i].signedPassword := 'ser';
						GVL_USER.user_array[i].userGropuNumber :=4;
                    ELSIF GVL_USER.newuserGroupNumber =4 THEN
                        GVL_USER.user_array[i].signedPassword := 'tech';
						GVL_USER.user_array[i].userGropuNumber :=5;
                    ELSIF GVL_USER.newuserGroupNumber =2 THEN
                        GVL_USER.user_array[i].signedPassword := 'mech';
						GVL_USER.user_array[i].userGropuNumber :=2;
                    END_IF
                    
                    // Potwierdzenie dodania nowego użytkownika
                    GVL_USER.new_user_added := TRUE;
                    GVL_USER.new_user_add_error := FALSE;
                    freeSlot := TRUE;  // Znalazło się wolne miejsce
					gvl_user.bwait := FALSE;
                    EXIT;  // Możemy zakończyć pętlę, bo użytkownik został dodany
                END_IF
            END_FOR
        ELSE
            // Hasło, RFID lub QR już istnieje - błąd dodawania użytkownika
            GVL_USER.new_user_add_error := TRUE;
			gvl_user.bwait := FALSE;
        END_IF
    END_IF

    // Jeśli nie znaleziono wolnego miejsca, ustawiamy błąd dodawania
    IF NOT freeSlot THEN
        GVL_USER.new_user_add_error := TRUE;
		gvl_user.bwait := FALSE;
    END_IF
	GVL_USER.new_user:=FALSE;
	validGroup:=FALSE;
	GVL_USER.user_succesed_log := FALSE;
END_IF

IF NOT GVL_USER.new_user THEN
	GVL_USER.new_user_accept:=FALSE;
	gvl_user.bwait := FALSE;
	validGroup:=FALSE;
	GVL_USER.newpasswordQR:='';
	GVL_USER.newpasswordRFID:='';
	newuserLogoffbetween:='';
END_IF



// Edycja istniejącego użytkownika
IF GVL_USER.edit_user AND GVL_USER.edit_user_accept THEN
    GVL_USER.user_eddited := FALSE;
    GVL_USER.edit_user_error := TRUE;
    validGroup := FALSE;  // Na początku zakładamy, że grupa nie jest poprawna
	gvl_user.bwait := TRUE;
    
    // Sprawdzanie, czy użytkownik o podanym imieniu i nazwisku istnieje
    userExists := FALSE;
    FOR i := 1 TO 100 DO
        IF GVL_USER.user_array[i].enabled AND 
           GVL_USER.user_array[i].userNameSurname = GVL_USER.actual_editted_user THEN
            GVL_USER.currentUser := i;
            userExists := TRUE;
            EXIT;  // Zatrzymujemy pętlę, gdy znajdziemy użytkownika
        END_IF
    END_FOR

    // Jeśli użytkownik nie istnieje, kończymy edycję
    IF NOT userExists THEN
        GVL_USER.edit_user_error := TRUE;
        gvl_user.bwait := FALSE;
    ELSE
        // Sprawdzanie, czy użytkownik do edycji jest aktywny
        IF GVL_USER.user_array[GVL_USER.currentUser].enabled THEN
            // Aktualizacja danych użytkownika	

            // Sprawdzanie, czy Imię i Nazwisko ma być zmienione
            IF GVL_USER.edituserNameSurname <> "" THEN
                GVL_USER.user_array[GVL_USER.currentUser].userNameSurname := GVL_USER.edituserNameSurname;
            END_IF
			
            // Sprawdzanie, czy hasło ma być zmienione
			IF GVL_USER.editpassword <> '' THEN
                GVL_USER.user_array[GVL_USER.currentUser].password := GVL_USER.editpassword;
            END_IF

            // Sprawdzanie, czy RFID ma być zmienione
            IF GVL_USER.editpasswordRFID <> '' THEN
                GVL_USER.user_array[GVL_USER.currentUser].passwordRFID := GVL_USER.editpasswordRFID;
            END_IF

            // Sprawdzanie, czy QR ma być zmienione
            IF GVL_USER.editpasswordQR <> '' THEN
                GVL_USER.user_array[GVL_USER.currentUser].passwordQR := GVL_USER.editpasswordQR;
            END_IF
			
			// Sprawdzanie, czy czas wylogowania ma być zmieniony
           // IF GVL_USER.editautoLogOff <> '' THEN
			//	edituserLogoffbetween := CONCAT('PT', GVL_USER.editautoLogOff);
           //     //GVL_USER.user_array[GVL_USER.currentUser].autoLogOff := CONCAT(edituserLogoffbetween, 'M');
           // END_IF

            // Sprawdzanie, czy grupa ma być zmieniona
            IF GVL_USER.edituserGroupNumber <> 0 THEN
                // Sprawdzanie, czy wybrana grupa jest jedną z dozwolonych
                FOR j := 1 TO 5 DO
                    IF GVL_USER.edituserGroupNumber = allowedGroupsnumber[j] THEN
                        validGroup := TRUE;  // Jeśli grupa jest dozwolona, ustawiamy na TRUE
                        EXIT;  // Wychodzimy z pętli, bo znaleźliśmy poprawną grupę
                    END_IF
                END_FOR

                // Jeśli grupa nie jest poprawna, przerywamy proces edycji użytkownika
                IF NOT validGroup THEN
                    GVL_USER.edit_user_error := TRUE;
					gvl_user.bwait := FALSE;
					RETURN;  // Kończymy operację, gdy grupa jest nieprawidłowa
                ELSE
                    GVL_USER.user_array[GVL_USER.currentUser].userGroup := GVL_USER.edituserGroup;
                END_IF
            END_IF
            
            // Potwierdzenie edycji użytkownika
            GVL_USER.user_eddited := TRUE;
            GVL_USER.edit_user_error := FALSE;
			gvl_user.bwait := FALSE;
			GVL_USER.user_succesed_log := FALSE;
        END_IF
    END_IF
END_IF

IF NOT GVL_USER.edit_user THEN
	GVL_USER.edit_user_accept:=FALSE;
	gvl_user.bwait := FALSE;
END_IF


// Usuwanie użytkownika
IF GVL_USER.delete_user AND GVL_USER.delete_user_accept THEN
    GVL_USER.delete_user_error := TRUE;  // Zakładamy na początku, że operacja się nie uda
    GVL_USER.user_deleted_succes := FALSE;  // Zmienna sygnalizująca usunięcie użytkownika
    
    // Sprawdzanie, czy użytkownik o podanym imieniu i nazwisku istnieje
    userExists_2 := FALSE;
    FOR i := 1 TO 100 DO
        IF GVL_USER.user_array[i].enabled AND 
           GVL_USER.user_array[i].userNameSurname = GVL_USER.choosen_to_delete THEN
           
            // Użytkownik znaleziony, usuwamy go
            GVL_USER.user_array[i].userID := 0;
            //GVL_USER.user_array[i].domain := '';
            GVL_USER.user_array[i].enabled := FALSE;
            GVL_USER.user_array[i].userLogin := '';
            GVL_USER.user_array[i].userNameSurname := "";
            GVL_USER.user_array[i].password := '';
			GVL_USER.user_array[i].signedPassword := '';
            GVL_USER.user_array[i].passwordRFID := '';
            GVL_USER.user_array[i].passwordQR := '';
            GVL_USER.user_array[i].userGroup := '';
			GVL_USER.user_array[i].userGropuNumber:=0;
            //GVL_USER.user_array[i].autoLogOff := '';
           // GVL_USER.user_array[i].locale := '';
            //GVL_USER.user_array[i].timeFormatlocale := '';
           // GVL_USER.user_array[i].timeZone := '';
            
            userExists_2 := TRUE;
            GVL_USER.delete_user_error := FALSE;  // Operacja usunięcia powiodła się
            GVL_USER.user_deleted_succes := TRUE;  // Potwierdzenie, że użytkownik został usunięty
            EXIT;  // Zatrzymanie pętli po znalezieniu i usunięciu użytkownika
        END_IF
    END_FOR
    
    // Jeśli użytkownika nie znaleziono, ustaw błąd
    IF NOT userExists_2 THEN
        GVL_USER.delete_user_error := TRUE;  // Nie znaleziono użytkownika
        GVL_USER.user_deleted_succes := FALSE;
    END_IF
	gvl_user.choosen_to_delete:="";
	gvl_user.delete_user_accept:=FALSE;
	userExists_2:=FALSE;
	GVL_USER.user_succesed_log := FALSE;
	GVL_USER.user_deleted_succes := FALSE;
END_IF


// Proces wylogowania użytkownika
IF GVL_USER.logout THEN
    // Czyszczenie danych aktualnie zalogowanego użytkownika
    IF GVL_USER.currentUser >= 1 AND GVL_USER.currentUser <= 100 THEN
       
        // Ustawienie użytkownika "niezalogowany" z wiersza pod indeksem 6
        GVL_USER.currentUser := 6;
		gvl_user.currentUserName :="Niezalogowany Użytkownik";
		gvl_user.currentUserGroup :='Niezalogowany';
		gvl_user.currentUserGroupNumber :=0; //
        GVL_USER.user_succesed_log := TRUE;  // Potwierdzenie, że wylogowanie i logowanie zakończyły się sukcesem
        GVL_USER.logout := FALSE;  // Resetowanie sygnału wylogowania
		GVL_USER.putted_user_password:='';
    END_IF
	GVL_USER.user_succesed_log := FALSE;
END_IF

//Proces nadpisania użytkowników w razie utraty Persistent
IF gvl_user.b_rewrite_users_after_issues OR bFirstCycle 
	THEN
	//admin
	gvl_user.user_array[1].userID:=0;
	gvl_user.user_array[1].enabled:=TRUE;
	gvl_user.user_array[1].userGroup:='Admin';
	gvl_user.user_array[1].userNameSurname:="Administrator";
	gvl_user.user_array[1].password:='adm';
	gvl_user.user_array[1].passwordRFID:='adm';
	gvl_user.user_array[1].passwordQR:='адм';
	gvl_user.user_array[1].userLogin:='adm';
	gvl_user.user_array[1].signedPassword:='adm';
	gvl_user.user_array[1].userGropuNumber:=1;
	//serwis
	gvl_user.user_array[3].userID:=2;
	gvl_user.user_array[3].enabled:=TRUE;
	gvl_user.user_array[3].userGroup:='Serwis';
	gvl_user.user_array[3].userNameSurname:="Serwisant";
	gvl_user.user_array[3].password:='ser';
	gvl_user.user_array[3].passwordRFID:='ser';
	gvl_user.user_array[3].passwordQR:='сер';
	gvl_user.user_array[3].userLogin:='ser';
	gvl_user.user_array[3].signedPassword:='ser';
	gvl_user.user_array[3].userGropuNumber:=4;
	//technolog
	gvl_user.user_array[4].userID:=3;
	gvl_user.user_array[4].enabled:=TRUE;
	gvl_user.user_array[4].userGroup:='Technolog';
	gvl_user.user_array[4].userNameSurname:="Technolog";
	gvl_user.user_array[4].password:='tech';
	gvl_user.user_array[4].passwordRFID:='tech';
	gvl_user.user_array[4].passwordQR:='тех';
	gvl_user.user_array[4].userLogin:='tech';	
	gvl_user.user_array[4].signedPassword:='tech';
	gvl_user.user_array[4].userGropuNumber:=5;
	//operator
	gvl_user.user_array[2].userID:=1;
	gvl_user.user_array[2].enabled:=TRUE;
	gvl_user.user_array[2].userGroup:='Operator';
	gvl_user.user_array[2].userNameSurname:="Operator";
	gvl_user.user_array[2].password:='opr';
	gvl_user.user_array[2].passwordRFID:='opr';
	gvl_user.user_array[2].passwordQR:='опр';
	gvl_user.user_array[2].userLogin:='opr';	
	gvl_user.user_array[2].signedPassword:='opr';
	gvl_user.user_array[2].userGropuNumber:=3;
	//mechanik
	gvl_user.user_array[5].userID:=4;
	gvl_user.user_array[5].enabled:=TRUE;
	gvl_user.user_array[5].userGroup:='Mechanik';
	gvl_user.user_array[5].userNameSurname:="Mechanik";
	gvl_user.user_array[5].password:='mech';
	gvl_user.user_array[5].passwordRFID:='mech';
	gvl_user.user_array[5].passwordQR:='мех';
	gvl_user.user_array[5].userLogin:='mech';	
	gvl_user.user_array[5].signedPassword:='mech';
	gvl_user.user_array[5].userGropuNumber:=2;
	//Tymur
	gvl_user.user_array[7].userID:=7;
	gvl_user.user_array[7].enabled:=TRUE;
	gvl_user.user_array[7].userGroup:='Operator';
	gvl_user.user_array[7].userNameSurname:="Tymur Knis";
	gvl_user.user_array[7].password:='11031988';
	gvl_user.user_array[7].passwordRFID:='tup2';
	gvl_user.user_array[7].passwordQR:='tup2';
	gvl_user.user_array[7].userLogin:='11031988';	
	gvl_user.user_array[7].signedPassword:='opr';
	gvl_user.user_array[7].userGropuNumber:=3;
	//Dima
	gvl_user.user_array[8].userID:=8;
	gvl_user.user_array[8].enabled:=TRUE;
	gvl_user.user_array[8].userGroup:='Operator';
	gvl_user.user_array[8].userNameSurname:="Dima Mironenko";
	gvl_user.user_array[8].password:='023';
	gvl_user.user_array[8].passwordRFID:='tup1';
	gvl_user.user_array[8].passwordQR:='tup1';
	gvl_user.user_array[8].userLogin:='023';	
	gvl_user.user_array[8].signedPassword:='opr';
	gvl_user.user_array[8].userGropuNumber:=3;
	//Uruchomienie
	gvl_user.user_array[6].userID:=6;
	gvl_user.user_array[6].enabled:=TRUE;
	gvl_user.user_array[6].userGroup:='TKMATIK';
	gvl_user.user_array[6].userNameSurname:="TKMatik Uruchomienie";
	gvl_user.user_array[6].password:='parol';
	gvl_user.user_array[6].passwordRFID:='tup10';
	gvl_user.user_array[6].passwordQR:='tup10';
	gvl_user.user_array[6].userLogin:='parol';	
	gvl_user.user_array[6].signedPassword:='parol';
	gvl_user.user_array[6].userGropuNumber:=10;
	//odbiory
	gvl_user.user_array[9].userID:=9;
	gvl_user.user_array[9].enabled:=TRUE;
	gvl_user.user_array[9].userGroup:='Technolog';
	gvl_user.user_array[9].userNameSurname:="Odbiory";
	gvl_user.user_array[9].password:='odb';
	gvl_user.user_array[9].passwordRFID:='tup11';
	gvl_user.user_array[9].passwordQR:='tup11';
	gvl_user.user_array[9].userLogin:='odb';	
	gvl_user.user_array[9].signedPassword:='tech';
	gvl_user.user_array[9].userGropuNumber:=5;
END_IF

END_PROGRAM

// ---- POUs/DataLogging/P_Recipebackup.TcPOU
PROGRAM P_Recipebackup
VAR
	tonBackup : TON;                     // Timer TON 2 sekund
    tonHour : TON;                       // Timer TON 1 godzina
    bBackupActive : BOOL := FALSE;       // Flaga true
END_VAR

tonHour(IN := NOT tonHour.Q, PT := T#3600S);
IF tonHour.Q THEN
    // Zakończenie liczenia godziny, zaczynamy generowanie sygnału TRUE
    tonHour(IN := FALSE);                // Zresetuj timer godziny
    bBackupActive := TRUE;               // Aktywuj sygnał TRUE
    tonBackup(IN := TRUE, PT := T#2S);   // Zainicjuj timer na 2 sekundy
END_IF

// Timer dla 2 sekundowego sygnału
IF tonBackup.Q THEN
    bBackupActive := FALSE;              // Wyłącz sygnał TRUE po 2 sekundach
    tonBackup(IN := FALSE);              // Zresetuj timer backupu
END_IF
gvl_recipe.b_recipe_backup := bBackupActive;

END_PROGRAM

// ---- POUs/DataLogging/P_Gauge_Measures.TcPOU
PROGRAM P_Gauge_Measures
VAR
	lr_receaved_weight_from_recipe :LREAL;
	lr_max_value :LREAL;
	
	lr_tolerance_actual_low :LREAL;
	lr_tolerance_actual_high :LREAL;
	lr_tolerance_actual_low_weight :LREAL;
	lr_tolerance_actual_high_weight :LREAL;
	
	lr_measured_weight_1 :LREAL;
	s_measured_weight_1_show :STRING;
	s_difference_weight_1_show :STRING;
	lr_difference_weight_1_show_math :LREAL;
	lr_measured_weight_2 :LREAL;
	s_measured_weight_2_show :STRING;
	s_difference_weight_2_show :STRING;
	lr_difference_weight_2_show_math :LREAL;
	lr_measured_weight_3 :LREAL;
	s_measured_weight_3_show :STRING;
	s_difference_weight_3_show :STRING;
	lr_difference_weight_3_show_math :LREAL;
	lr_measured_weight_4 :LREAL;
	s_difference_weight_4_show :STRING;
	s_measured_weight_4_show :STRING;
	lr_difference_weight_4_show_math :LREAL;
	
	s_correction_weight_1	:STRING;
	lr_correction_weight_1_math	:LREAL;
	s_correction_weight_2	:STRING;
	lr_correction_weight_2_math	:LREAL;	
	s_correction_weight_3	:STRING;
	lr_correction_weight_3_math	:LREAL;
	s_correction_weight_4	:STRING;
	lr_correction_weight_4_math	:LREAL;
	
	lr_dosed_1_math			:LREAL;
	s_dosed_1				:STRING;
	lr_dosed_2_math			:LREAL;
	s_dosed_2				:STRING;	
	lr_dosed_3_math			:LREAL;
	s_dosed_3				:STRING;
	lr_dosed_4_math			:LREAL;
	s_dosed_4				:STRING;
	
//korekta	
	lr_add_correction_value_1	:LREAL;
	lr_add_correction_value_2	:LREAL;
	lr_add_correction_value_3	:LREAL;
	lr_add_correction_value_4	:LREAL;
	lr_sub_correction_value_1	:LREAL;
	lr_sub_correction_value_2	:LREAL;
	lr_sub_correction_value_3	:LREAL;
	lr_sub_correction_value_4	:LREAL;	
	
//zakręcanie	
	lr_torque_recipe_set		:LREAL;
	lr_torque_recipe_set_2		:LREAL;
	lr_torque_1					:LREAL;
	s_torque_1					:STRING;
	lr_torque_2					:LREAL;
	s_torque_2					:STRING;
	lr_torq_diff_1				:LREAL;
	lr_torq_diff_2				:LREAL;
	s_torq_diff_1				:STRING;
	s_torq_diff_2				:STRING;
	lr_low_torque_1				:LREAL;
	lr_low_torque_2				:LREAL;
	lr_high_torque_1			:LREAL;
	lr_high_torque_2			:LREAL;
	
//poziomy w zbiornikach
	i_tank_lvl_1				:INT;
	s_tank_lvl_1				:STRING;
	i_tank_lvl_2				:INT;
	s_tank_lvl_2				:STRING;	
	lr_try_value				:lreal;
	
END_VAR

//maksymalny zakres miernika
lr_receaved_weight_from_recipe:=gvl_gauge.lr_WeightMass_recipe; //otrzymanie wartości z receptur
lr_max_value:=2*lr_receaved_weight_from_recipe; //zwiększenie zakresu maksymalnej wagi
gvl_gauge.lr_out_max_weight_value:=lr_max_value; //przepisanie wartości maksymalnej do wykresów wag

//tolerancje dozowników
lr_tolerance_actual_low_weight:=gvl_gauge.lr_Tolerance_Low; //przepisanie wartości z receptury
lr_tolerance_actual_high_weight:=gvl_gauge.lr_Tolerance_High; //przepisanie wartości z receptury
lr_tolerance_actual_low:=lr_receaved_weight_from_recipe-lr_tolerance_actual_low_weight; //ustalenie dolnej granicy
lr_tolerance_actual_high:=lr_receaved_weight_from_recipe+lr_tolerance_actual_high_weight; //ustalenie górnej granicy 
gvl_gauge.lr_out_min_tolerance_low:=lr_tolerance_actual_low; //przepisanie dolnej granicy
gvl_gauge.lr_out_max_tolerance_high:=lr_tolerance_actual_high; //przepisanie górnej granicy 

//powiększenie wskazania pomiaru
lr_measured_weight_1:=p_ads_gauge.lr_weight_1;
lr_measured_weight_2:=p_ads_gauge.lr_weight_2;
lr_measured_weight_3:=p_ads_gauge.lr_weight_3;
lr_measured_weight_4:=p_ads_gauge.lr_weight_4;

//wskazanie w lewym rogu aktualnej wagi
s_measured_weight_1_show:=CONCAT(LREAL_TO_STRING((TRUNC(p_ads_gauge.lr_weight_1 * 10))/10.0),' g');
s_measured_weight_2_show:=CONCAT(LREAL_TO_STRING((TRUNC(p_ads_gauge.lr_weight_2 * 10))/10.0),' g');
s_measured_weight_3_show:=CONCAT(LREAL_TO_STRING((TRUNC(p_ads_gauge.lr_weight_3 * 10))/10.0),' g');
s_measured_weight_4_show:=CONCAT(LREAL_TO_STRING((TRUNC(p_ads_gauge.lr_weight_4 * 10))/10.0),' g');
	
IF NOT gvl_gauge.bDosingTwoPhasesShow THEN	
	gvl_gauge.s_actual_weight_1:=concat(LREAL_TO_fmtstr(lr_measured_weight_1,1,TRUE), ' g');
	gvl_gauge.s_actual_weight_2:=concat(LREAL_TO_fmtstr(lr_measured_weight_2,1,TRUE), ' g');
	gvl_gauge.s_actual_weight_3:=concat(LREAL_TO_fmtstr(lr_measured_weight_3,1,TRUE), ' g');
	gvl_gauge.s_actual_weight_4:=concat(LREAL_TO_fmtstr(lr_measured_weight_4,1,TRUE), ' g');
ELSE	
	gvl_gauge.s_actual_weight_1:=concat(LREAL_TO_fmtstr(lr_receaved_weight_from_recipe,1,TRUE), ' g');		
    gvl_gauge.s_actual_weight_2:=concat(LREAL_TO_fmtstr(lr_receaved_weight_from_recipe,1,TRUE), ' g');
    gvl_gauge.s_actual_weight_3:=concat(LREAL_TO_fmtstr(lr_receaved_weight_from_recipe,1,TRUE), ' g');
    gvl_gauge.s_actual_weight_4:=concat(LREAL_TO_fmtstr(lr_receaved_weight_from_recipe,1,TRUE), ' g');
END_IF
	
	//wskazanie różnicy pomiaru w prawym rogu
	lr_difference_weight_1_show_math:=lr_receaved_weight_from_recipe - p_ads_gauge.lr_weight_1;
	s_difference_weight_1_show:=CONCAT((LREAL_TO_FMTSTR(lr_difference_weight_1_show_math,1,TRUE)),' g');
	
	lr_difference_weight_2_show_math:=lr_receaved_weight_from_recipe - p_ads_gauge.lr_weight_2;
	s_difference_weight_2_show:=CONCAT((LREAL_TO_FMTSTR(lr_difference_weight_2_show_math,1,TRUE)),' g');
	
	lr_difference_weight_3_show_math:=lr_receaved_weight_from_recipe - p_ads_gauge.lr_weight_3;
	s_difference_weight_3_show:=CONCAT((LREAL_TO_FMTSTR(lr_difference_weight_3_show_math,1,TRUE)),' g');
	
	lr_difference_weight_4_show_math:=lr_receaved_weight_from_recipe - p_ads_gauge.lr_weight_4;
	s_difference_weight_4_show:=CONCAT((LREAL_TO_FMTSTR(lr_difference_weight_4_show_math,1,TRUE)),' g');

If NOT gvl_gauge.bDosingTwoPhasesShow then	
	gvl_gauge.s_actual_weight_1_diff:=s_difference_weight_1_show;
	gvl_gauge.s_actual_weight_2_diff:=s_difference_weight_2_show;
	gvl_gauge.s_actual_weight_3_diff:=s_difference_weight_3_show;
	gvl_gauge.s_actual_weight_4_diff:=s_difference_weight_4_show;
ELSE
	gvl_gauge.s_actual_weight_1_diff:= '0';	
    gvl_gauge.s_actual_weight_2_diff:= '0';
    gvl_gauge.s_actual_weight_3_diff:= '0';
    gvl_gauge.s_actual_weight_4_diff:= '0';
END_IF

//wyświetlanie korekty prawy górny róg
lr_correction_weight_1_math:=p_ads_gauge.lr_correction_weight_1;
s_correction_weight_1:=concat(LREAL_TO_fmtstr(lr_correction_weight_1_math,1,TRUE), ' ml');

lr_correction_weight_2_math:=p_ads_gauge.lr_correction_weight_2;
s_correction_weight_2:=concat(LREAL_TO_fmtstr(lr_correction_weight_2_math,1,TRUE), ' ml');

lr_correction_weight_3_math:=p_ads_gauge.lr_correction_weight_3;
s_correction_weight_3:=concat(LREAL_TO_fmtstr(lr_correction_weight_3_math,1,TRUE), ' ml');

lr_correction_weight_4_math:=p_ads_gauge.lr_correction_weight_4;
s_correction_weight_4:=concat(LREAL_TO_fmtstr(lr_correction_weight_4_math,1,TRUE), ' ml');


gvl_gauge.s_actual_corr_1:=s_correction_weight_1;
gvl_gauge.s_actual_corr_2:=s_correction_weight_2;
gvl_gauge.s_actual_corr_3:=s_correction_weight_3;
gvl_gauge.s_actual_corr_4:=s_correction_weight_4;

//wyświetlanie wydozowanej ilości lewy górny róg
s_dosed_1:=concat(LREAL_TO_fmtstr(p_ads_gauge.lr_dosed_1,1,TRUE),' ml');

s_dosed_2:=concat(LREAL_TO_fmtstr(p_ads_gauge.lr_dosed_2,1,TRUE),' ml');

s_dosed_3:=concat(LREAL_TO_fmtstr(p_ads_gauge.lr_dosed_3,1,TRUE),' ml');

s_dosed_4:=concat(LREAL_TO_fmtstr(p_ads_gauge.lr_dosed_4,1,TRUE),' ml');

gvl_gauge.s_actual_dose_1:=s_dosed_1;
gvl_gauge.s_actual_dose_2:=s_dosed_2;
gvl_gauge.s_actual_dose_3:=s_dosed_3;
gvl_gauge.s_actual_dose_4:=s_dosed_4;

//zmiana korekty dozowania
lr_add_correction_value_1:=lr_correction_weight_1_math+0.5;
lr_add_correction_value_2:=lr_correction_weight_2_math+0.5;
lr_add_correction_value_3:=lr_correction_weight_3_math+0.5;
lr_add_correction_value_4:=lr_correction_weight_4_math+0.5;

lr_sub_correction_value_1:=lr_correction_weight_1_math-0.5;
lr_sub_correction_value_2:=lr_correction_weight_2_math-0.5;
lr_sub_correction_value_3:=lr_correction_weight_3_math-0.5;
lr_sub_correction_value_4:=lr_correction_weight_4_math-0.5;

gvl_gauge.lr_corr_add_1:=lr_add_correction_value_1;
gvl_gauge.lr_corr_add_2:=lr_add_correction_value_2;
gvl_gauge.lr_corr_add_3:=lr_add_correction_value_3;
gvl_gauge.lr_corr_add_4:=lr_add_correction_value_4;
gvl_gauge.lr_corr_sub_1:=lr_sub_correction_value_1;
gvl_gauge.lr_corr_sub_2:=lr_sub_correction_value_2;
gvl_gauge.lr_corr_sub_3:=lr_sub_correction_value_3;
gvl_gauge.lr_corr_sub_4:=lr_sub_correction_value_4;

//momenty i różnice
lr_torque_recipe_set:=p_ads_gauge.lr_screwer_torque_set;
lr_torque_recipe_set_2:=p_ads_gauge.lr_screwer_torque_set_2;
lr_torque_1:=p_ads_gauge.lr_screwer_torque_1;
s_torque_1:=concat(LREAL_TO_fmtstr(lr_torque_1,1,TRUE),' Nm');
gvl_gauge.s_actual_torque_1:=s_torque_1;
lr_torque_2:=p_ads_gauge.lr_screwer_torque_2;
s_torque_2:=concat(LREAL_TO_fmtstr(lr_torque_2,1,TRUE),' Nm');
gvl_gauge.s_actual_torque_2:=s_torque_2;

lr_torq_diff_1:=lr_torque_recipe_set - lr_torque_1;
s_torq_diff_1:=concat(LREAL_TO_FMTSTR(lr_torq_diff_1,1,TRUE),' Nm');
gvl_gauge.s_actual_torque_diff_1:=s_torq_diff_1;
lr_torq_diff_2:=lr_torque_recipe_set_2 - lr_torque_2;
s_torq_diff_2:=concat(LREAL_TO_FMTSTR(lr_torq_diff_2,1,TRUE),' Nm');
gvl_gauge.s_actual_torque_diff_2:=s_torq_diff_2;


gvl_gauge.lr_out_torque_high_1:=lr_torque_recipe_set*1.1;
gvl_gauge.lr_out_torque_high_2:=lr_torque_recipe_set_2*1.1;
gvl_gauge.lr_out_torque_low_1:=lr_torque_recipe_set*0.9;
gvl_gauge.lr_out_torque_low_2:=lr_torque_recipe_set_2*0.9;


//poziomy zbiorników
i_tank_lvl_1:=p_ads_gauge.isensor_value_1;
s_tank_lvl_1:=concat(INT_TO_STRING(i_tank_lvl_1),' mm');
gvl_gauge.s_actual_level_1:=s_tank_lvl_1;
i_tank_lvl_2:=p_ads_gauge.isensor_value_2;
s_tank_lvl_2:=concat(INT_TO_STRING(i_tank_lvl_2),' mm');
gvl_gauge.s_actual_level_2:=s_tank_lvl_2;

IF NOT gvl_gauge.bDosingTwoPhasesShow THEN	
	gvl_gauge.lr_out_weight_measured_1	:=	lr_measured_weight_1;
	gvl_gauge.lr_out_weight_measured_2	:=	lr_measured_weight_2;
	gvl_gauge.lr_out_weight_measured_3	:=	lr_measured_weight_3;
	gvl_gauge.lr_out_weight_measured_4	:=	lr_measured_weight_4;
ELSE                                  	
	gvl_gauge.lr_out_weight_measured_1	:=	lr_receaved_weight_from_recipe;
    gvl_gauge.lr_out_weight_measured_2	:=	lr_receaved_weight_from_recipe;
    gvl_gauge.lr_out_weight_measured_3	:=	lr_receaved_weight_from_recipe;
    gvl_gauge.lr_out_weight_measured_4	:=	lr_receaved_weight_from_recipe;
END_IF

gvl_gauge.s_out_weight_measured_1:=concat(LREAL_TO_fmtstr(lr_measured_weight_1,1,TRUE), ' g');
gvl_gauge.s_out_weight_measured_2:=concat(LREAL_TO_fmtstr(lr_measured_weight_2,1,TRUE), ' g');
gvl_gauge.s_out_weight_measured_3:=concat(LREAL_TO_fmtstr(lr_measured_weight_3,1,TRUE), ' g');
gvl_gauge.s_out_weight_measured_4:=concat(LREAL_TO_fmtstr(lr_measured_weight_4,1,TRUE), ' g');


gvl_gauge.lr_diff_dispencer_2:=	P_ads_gauge.lrDispencer2DoseVolumeShow-P_ads_gauge.lrDispencer2Phase1VolumeShow-P_ads_gauge.lrDispencer2Phase2VolumeShow;
gvl_gauge.lr_diff_dispencer_1:= P_ads_gauge.lrDispencer1DoseVolumeShow-P_ads_gauge.lrDispencer1Phase1VolumeShow-P_ads_gauge.lrDispencer1Phase2VolumeShow;

END_PROGRAM

// ---- POUs/ADS/P_ADS_Gauge.TcPOU
PROGRAM P_ADS_Gauge
VAR
	bTrigger				: BOOL;
	lr_weight_1				:LREAL;
	lr_weight_2				:LREAL;
	lr_weight_3				:LREAL;
	lr_weight_4				:LREAL;
	
	lr_correction_weight_1  :LREAL;
	lr_correction_weight_2  :LREAL;
	lr_correction_weight_3  :LREAL;
	lr_correction_weight_4  :LREAL;	
	
	lr_dosed_1				:LREAL;
	lr_dosed_2				:LREAL;
	lr_dosed_3				:LREAL;
	lr_dosed_4				:LREAL;
	
	isensor_value_1			:INT;
	isensor_value_2			:INT;
	
	lr_screwer_torque_1		:LREAL;
	lr_screwer_torque_2		:LREAL;
	lr_screwer_torque_set	:LREAL;
	lr_screwer_torque_set_2	:LREAL;
//weight measureg
	fbRead_1: FB_ReadAdsSymByName;
	fbRead_2: FB_ReadAdsSymByName;
	fbRead_3: FB_ReadAdsSymByName;
	fbRead_4: FB_ReadAdsSymByName;
//correction weight	
	fbRead_5: FB_ReadAdsSymByName;
	fbRead_6: FB_ReadAdsSymByName;
	fbRead_7: FB_ReadAdsSymByName;
	fbRead_8: FB_ReadAdsSymByName;
//dose volume
	fbRead_9: FB_ReadAdsSymByName;
	fbRead_10: FB_ReadAdsSymByName;
	fbRead_11: FB_ReadAdsSymByName;
	fbRead_12: FB_ReadAdsSymByName;
//tank level
	fbRead_13: FB_ReadAdsSymByName;
	fbRead_14: FB_ReadAdsSymByName;
//Screwer torque
	fbRead_17: FB_ReadAdsSymByName;
	fbRead_16: FB_ReadAdsSymByName;
//Screwer torque recipe
	fbRead_15: FB_ReadAdsSymByName;
	fbRead_18: FB_ReadAdsSymByName;
	
	fbCyclicReadout: TON;
	//dispencer diff
	fbRead_19: FB_ReadAdsSymByName;
	fbRead_20: FB_ReadAdsSymByName;
	fbRead_21: FB_ReadAdsSymByName;
	
	fbRead_22: FB_ReadAdsSymByName;
	fbRead_23: FB_ReadAdsSymByName;
	fbRead_24: FB_ReadAdsSymByName;	
	
	lrDispencer2DoseVolumeShow:LREAL;
	lrDispencer2Phase1VolumeShow:LREAL;
	lrDispencer2Phase2VolumeShow:LREAL;
	lrDispencer1DoseVolumeShow:LREAL;
	lrDispencer1Phase1VolumeShow:LREAL;
	lrDispencer1Phase2VolumeShow:LREAL;
	
	
	fbRead_25: FB_ReadAdsSymByName;
	fbRead_26: FB_ReadAdsSymByName;
	fbRead_27: FB_ReadAdsSymByName;
	fbRead_28: FB_ReadAdsSymByName;
END_VAR

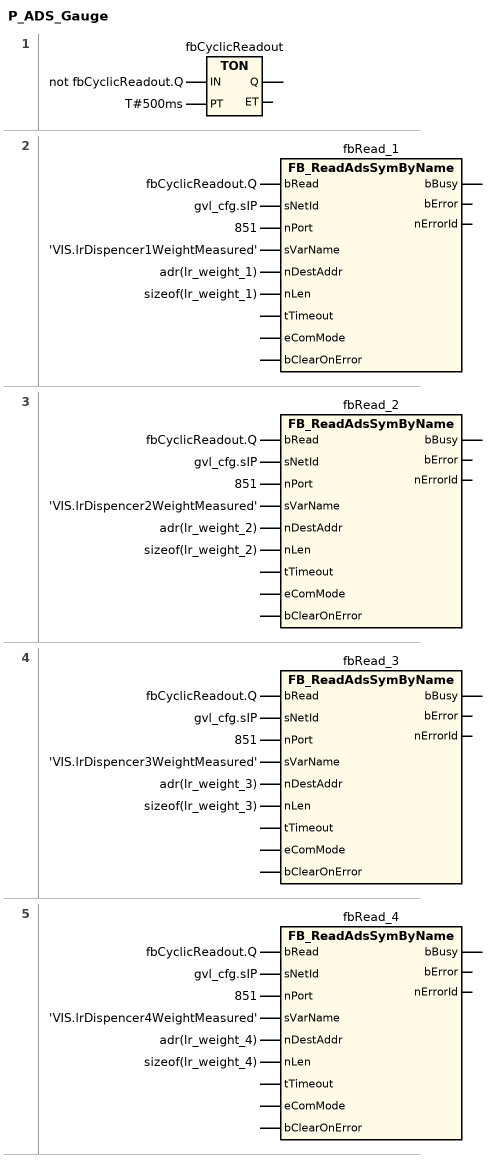
// NETWORK 1
fbCyclicReadout(IN := not fbCyclicReadout.Q, PT := T#500ms); // TON

// NETWORK 2
fbRead_1(
    bRead := fbCyclicReadout.Q,
    sNetId := gvl_cfg.sIP,
    nPort := 851,
    sVarName := 'VIS.lrDispencer1WeightMeasured',
    nDestAddr := adr(lr_weight_1),
    nLen := sizeof(lr_weight_1)); // FB_ReadAdsSymByName

// NETWORK 3
fbRead_2(
    bRead := fbCyclicReadout.Q,
    sNetId := gvl_cfg.sIP,
    nPort := 851,
    sVarName := 'VIS.lrDispencer2WeightMeasured',
    nDestAddr := adr(lr_weight_2),
    nLen := sizeof(lr_weight_2)); // FB_ReadAdsSymByName

// NETWORK 4
fbRead_3(
    bRead := fbCyclicReadout.Q,
    sNetId := gvl_cfg.sIP,
    nPort := 851,
    sVarName := 'VIS.lrDispencer3WeightMeasured',
    nDestAddr := adr(lr_weight_3),
    nLen := sizeof(lr_weight_3)); // FB_ReadAdsSymByName

// NETWORK 5
fbRead_4(
    bRead := fbCyclicReadout.Q,
    sNetId := gvl_cfg.sIP,
    nPort := 851,
    sVarName := 'VIS.lrDispencer4WeightMeasured',
    nDestAddr := adr(lr_weight_4),
    nLen := sizeof(lr_weight_4)); // FB_ReadAdsSymByName

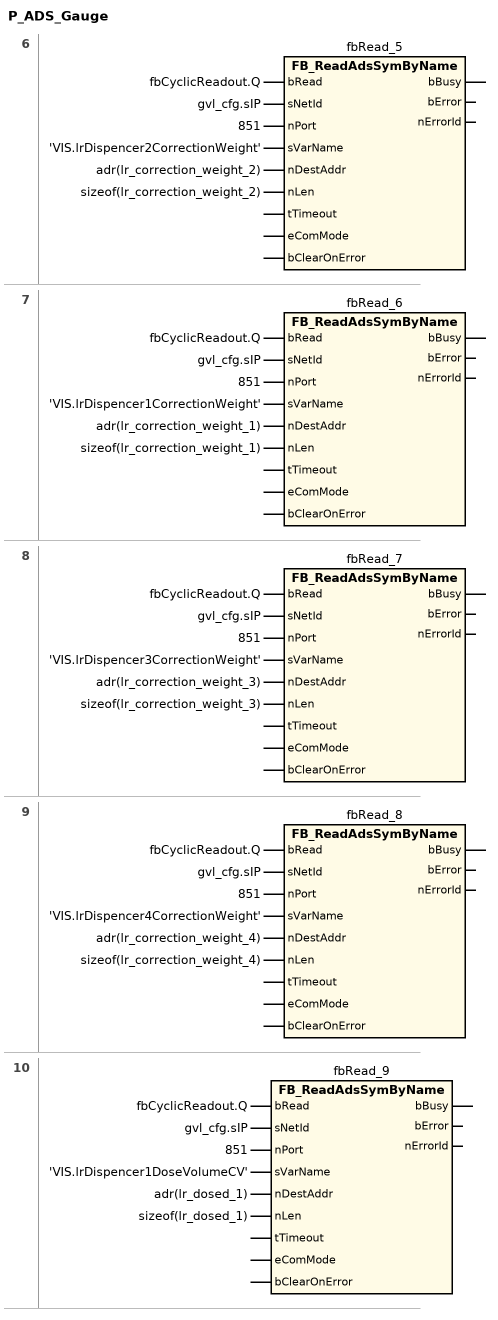
// NETWORK 6
fbRead_5(
    bRead := fbCyclicReadout.Q,
    sNetId := gvl_cfg.sIP,
    nPort := 851,
    sVarName := 'VIS.lrDispencer2CorrectionWeight',
    nDestAddr := adr(lr_correction_weight_2),
    nLen := sizeof(lr_correction_weight_2)); // FB_ReadAdsSymByName

// NETWORK 7
fbRead_6(
    bRead := fbCyclicReadout.Q,
    sNetId := gvl_cfg.sIP,
    nPort := 851,
    sVarName := 'VIS.lrDispencer1CorrectionWeight',
    nDestAddr := adr(lr_correction_weight_1),
    nLen := sizeof(lr_correction_weight_1)); // FB_ReadAdsSymByName

// NETWORK 8
fbRead_7(
    bRead := fbCyclicReadout.Q,
    sNetId := gvl_cfg.sIP,
    nPort := 851,
    sVarName := 'VIS.lrDispencer3CorrectionWeight',
    nDestAddr := adr(lr_correction_weight_3),
    nLen := sizeof(lr_correction_weight_3)); // FB_ReadAdsSymByName

// NETWORK 9
fbRead_8(
    bRead := fbCyclicReadout.Q,
    sNetId := gvl_cfg.sIP,
    nPort := 851,
    sVarName := 'VIS.lrDispencer4CorrectionWeight',
    nDestAddr := adr(lr_correction_weight_4),
    nLen := sizeof(lr_correction_weight_4)); // FB_ReadAdsSymByName

// NETWORK 10
fbRead_9(
    bRead := fbCyclicReadout.Q,
    sNetId := gvl_cfg.sIP,
    nPort := 851,
    sVarName := 'VIS.lrDispencer1DoseVolumeCV',
    nDestAddr := adr(lr_dosed_1),
    nLen := sizeof(lr_dosed_1)); // FB_ReadAdsSymByName

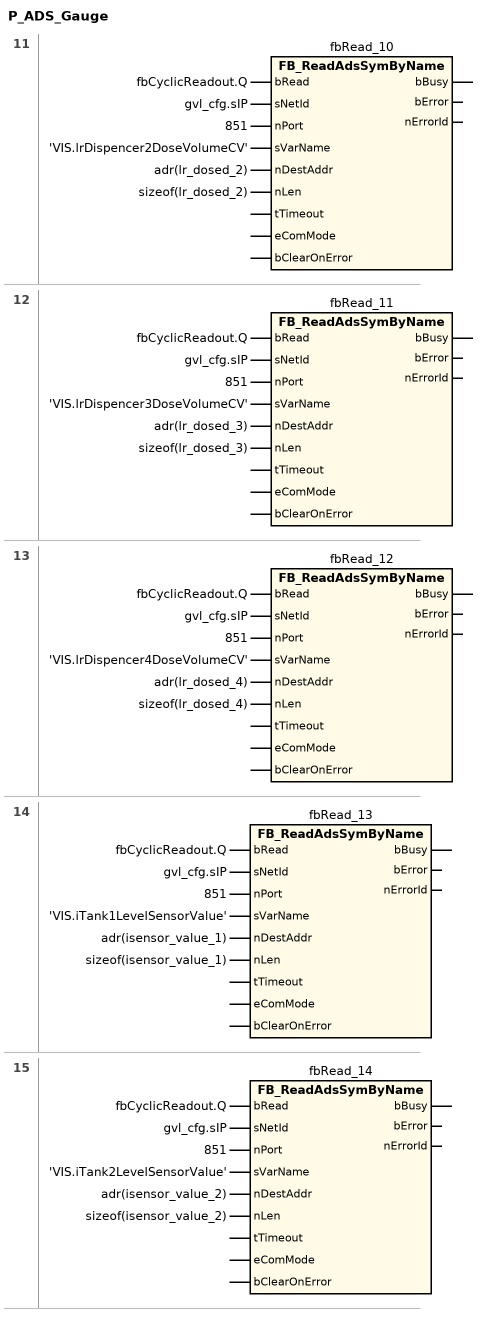
// NETWORK 11
fbRead_10(
    bRead := fbCyclicReadout.Q,
    sNetId := gvl_cfg.sIP,
    nPort := 851,
    sVarName := 'VIS.lrDispencer2DoseVolumeCV',
    nDestAddr := adr(lr_dosed_2),
    nLen := sizeof(lr_dosed_2)); // FB_ReadAdsSymByName

// NETWORK 12
fbRead_11(
    bRead := fbCyclicReadout.Q,
    sNetId := gvl_cfg.sIP,
    nPort := 851,
    sVarName := 'VIS.lrDispencer3DoseVolumeCV',
    nDestAddr := adr(lr_dosed_3),
    nLen := sizeof(lr_dosed_3)); // FB_ReadAdsSymByName

// NETWORK 13
fbRead_12(
    bRead := fbCyclicReadout.Q,
    sNetId := gvl_cfg.sIP,
    nPort := 851,
    sVarName := 'VIS.lrDispencer4DoseVolumeCV',
    nDestAddr := adr(lr_dosed_4),
    nLen := sizeof(lr_dosed_4)); // FB_ReadAdsSymByName

// NETWORK 14
fbRead_13(
    bRead := fbCyclicReadout.Q,
    sNetId := gvl_cfg.sIP,
    nPort := 851,
    sVarName := 'VIS.iTank1LevelSensorValue',
    nDestAddr := adr(isensor_value_1),
    nLen := sizeof(isensor_value_1)); // FB_ReadAdsSymByName

// NETWORK 15
fbRead_14(
    bRead := fbCyclicReadout.Q,
    sNetId := gvl_cfg.sIP,
    nPort := 851,
    sVarName := 'VIS.iTank2LevelSensorValue',
    nDestAddr := adr(isensor_value_2),
    nLen := sizeof(isensor_value_2)); // FB_ReadAdsSymByName

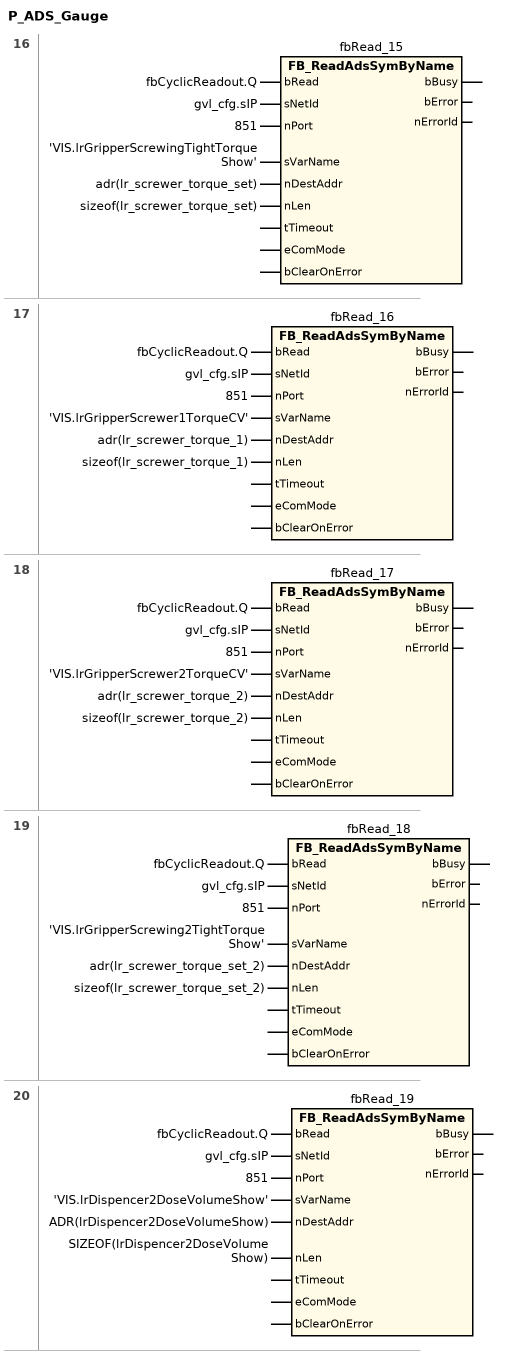
// NETWORK 16
fbRead_15(
    bRead := fbCyclicReadout.Q,
    sNetId := gvl_cfg.sIP,
    nPort := 851,
    sVarName := 'VIS.lrGripperScrewingTightTorqueShow',
    nDestAddr := adr(lr_screwer_torque_set),
    nLen := sizeof(lr_screwer_torque_set)); // FB_ReadAdsSymByName

// NETWORK 17
fbRead_16(
    bRead := fbCyclicReadout.Q,
    sNetId := gvl_cfg.sIP,
    nPort := 851,
    sVarName := 'VIS.lrGripperScrewer1TorqueCV',
    nDestAddr := adr(lr_screwer_torque_1),
    nLen := sizeof(lr_screwer_torque_1)); // FB_ReadAdsSymByName

// NETWORK 18
fbRead_17(
    bRead := fbCyclicReadout.Q,
    sNetId := gvl_cfg.sIP,
    nPort := 851,
    sVarName := 'VIS.lrGripperScrewer2TorqueCV',
    nDestAddr := adr(lr_screwer_torque_2),
    nLen := sizeof(lr_screwer_torque_2)); // FB_ReadAdsSymByName

// NETWORK 19
fbRead_18(
    bRead := fbCyclicReadout.Q,
    sNetId := gvl_cfg.sIP,
    nPort := 851,
    sVarName := 'VIS.lrGripperScrewing2TightTorqueShow',
    nDestAddr := adr(lr_screwer_torque_set_2),
    nLen := sizeof(lr_screwer_torque_set_2)); // FB_ReadAdsSymByName

// NETWORK 20
fbRead_19(
    bRead := fbCyclicReadout.Q,
    sNetId := gvl_cfg.sIP,
    nPort := 851,
    sVarName := 'VIS.lrDispencer2DoseVolumeShow',
    nDestAddr := ADR(lrDispencer2DoseVolumeShow),
    nLen := SIZEOF(lrDispencer2DoseVolumeShow)); // FB_ReadAdsSymByName

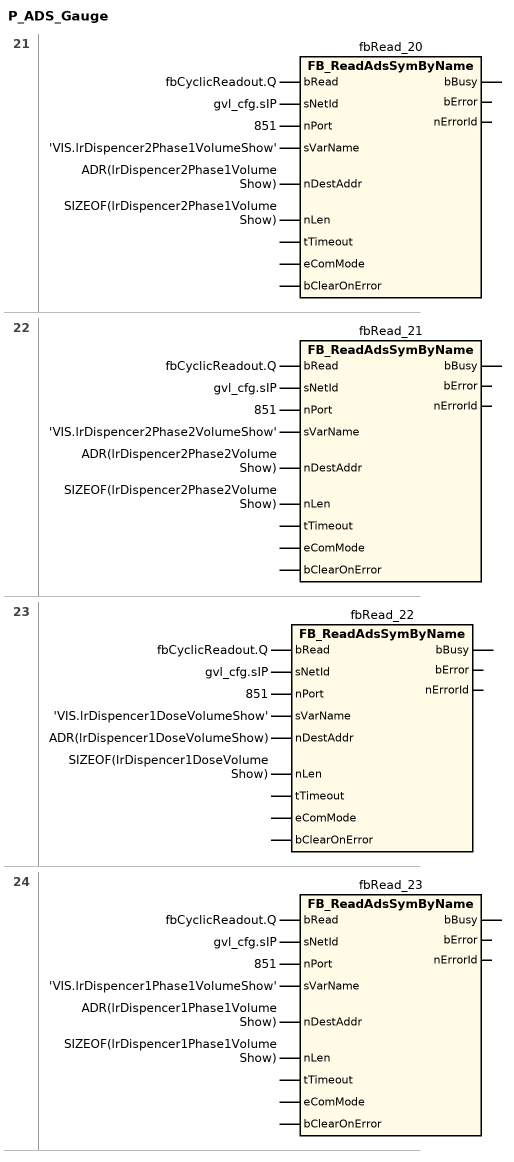
// NETWORK 21
fbRead_20(
    bRead := fbCyclicReadout.Q,
    sNetId := gvl_cfg.sIP,
    nPort := 851,
    sVarName := 'VIS.lrDispencer2Phase1VolumeShow',
    nDestAddr := ADR(lrDispencer2Phase1VolumeShow),
    nLen := SIZEOF(lrDispencer2Phase1VolumeShow)); // FB_ReadAdsSymByName

// NETWORK 22
fbRead_21(
    bRead := fbCyclicReadout.Q,
    sNetId := gvl_cfg.sIP,
    nPort := 851,
    sVarName := 'VIS.lrDispencer2Phase2VolumeShow',
    nDestAddr := ADR(lrDispencer2Phase2VolumeShow),
    nLen := SIZEOF(lrDispencer2Phase2VolumeShow)); // FB_ReadAdsSymByName

// NETWORK 23
fbRead_22(
    bRead := fbCyclicReadout.Q,
    sNetId := gvl_cfg.sIP,
    nPort := 851,
    sVarName := 'VIS.lrDispencer1DoseVolumeShow',
    nDestAddr := ADR(lrDispencer1DoseVolumeShow),
    nLen := SIZEOF(lrDispencer1DoseVolumeShow)); // FB_ReadAdsSymByName

// NETWORK 24
fbRead_23(
    bRead := fbCyclicReadout.Q,
    sNetId := gvl_cfg.sIP,
    nPort := 851,
    sVarName := 'VIS.lrDispencer1Phase1VolumeShow',
    nDestAddr := ADR(lrDispencer1Phase1VolumeShow),
    nLen := SIZEOF(lrDispencer1Phase1VolumeShow)); // FB_ReadAdsSymByName

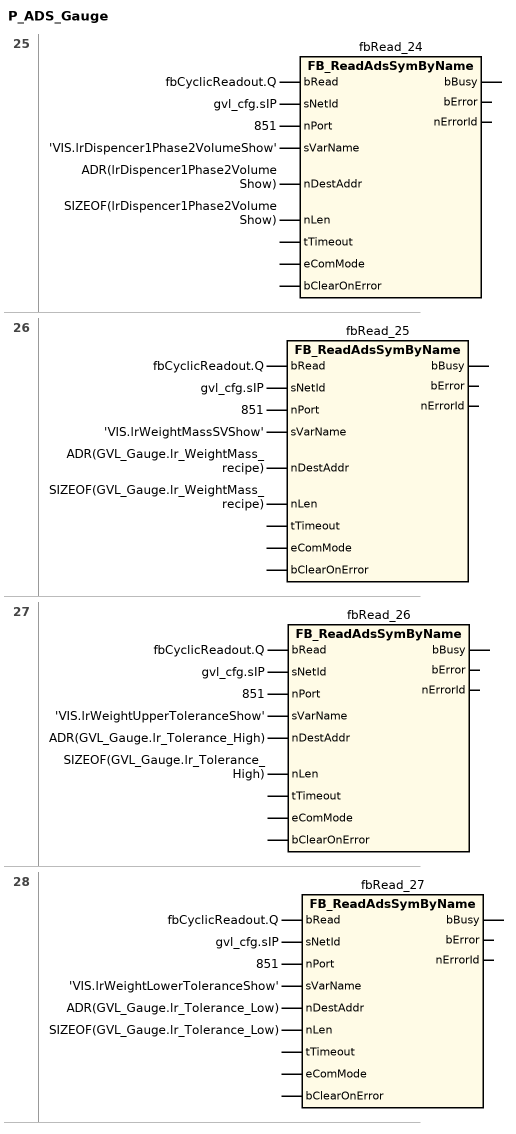
// NETWORK 25
fbRead_24(
    bRead := fbCyclicReadout.Q,
    sNetId := gvl_cfg.sIP,
    nPort := 851,
    sVarName := 'VIS.lrDispencer1Phase2VolumeShow',
    nDestAddr := ADR(lrDispencer1Phase2VolumeShow),
    nLen := SIZEOF(lrDispencer1Phase2VolumeShow)); // FB_ReadAdsSymByName

// NETWORK 26
fbRead_25(
    bRead := fbCyclicReadout.Q,
    sNetId := gvl_cfg.sIP,
    nPort := 851,
    sVarName := 'VIS.lrWeightMassSVShow',
    nDestAddr := ADR(GVL_Gauge.lr_WeightMass_recipe),
    nLen := SIZEOF(GVL_Gauge.lr_WeightMass_recipe)); // FB_ReadAdsSymByName

// NETWORK 27
fbRead_26(
    bRead := fbCyclicReadout.Q,
    sNetId := gvl_cfg.sIP,
    nPort := 851,
    sVarName := 'VIS.lrWeightUpperToleranceShow',
    nDestAddr := ADR(GVL_Gauge.lr_Tolerance_High),
    nLen := SIZEOF(GVL_Gauge.lr_Tolerance_High)); // FB_ReadAdsSymByName

// NETWORK 28
fbRead_27(
    bRead := fbCyclicReadout.Q,
    sNetId := gvl_cfg.sIP,
    nPort := 851,
    sVarName := 'VIS.lrWeightLowerToleranceShow',
    nDestAddr := ADR(GVL_Gauge.lr_Tolerance_Low),
    nLen := SIZEOF(GVL_Gauge.lr_Tolerance_Low)); // FB_ReadAdsSymByName

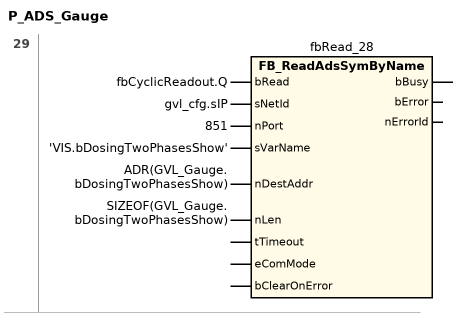
// NETWORK 29
fbRead_28(
    bRead := fbCyclicReadout.Q,
    sNetId := gvl_cfg.sIP,
    nPort := 851,
    sVarName := 'VIS.bDosingTwoPhasesShow',
    nDestAddr := ADR(GVL_Gauge.bDosingTwoPhasesShow),
    nLen := SIZEOF(GVL_Gauge.bDosingTwoPhasesShow)); // FB_ReadAdsSymByName

END_PROGRAM

// ---- POUs/DataLogging/P_RecipeChange.TcPOU
PROGRAM P_RecipeChange
VAR
	b_recipe_bool_change :R_trig;
	b_recipe_real_change :R_trig;
	b_recipe_was_changed_real :BOOL;
	b_recipe_was_changed_bool :BOOL;
	lr_old_param_bool :LREAL;
	lr_new_param_bool :LREAL;
	i :INT;
	nIndex      : INT := 0; 
    nTotalItems : INT := 500; 
	b_clear_recipe_history :BOOL:=FALSE;
END_VAR

b_recipe_bool_change(clk:= gvl_recipe.b_recipe_bool_change);
b_recipe_real_change(clk:= gvl_recipe.b_recipe_real_change);
b_clear_recipe_history:=FALSE;
IF gvl_recipe.b_recipe_real_change THEN //zmiana real
	IF (gvl_recipe.lr_recipe_change<>gvl_recipe.lr_recipe_change_1)  THEN
		b_recipe_was_changed_real:=TRUE;				
	END_IF
ELSE
	IF  gvl_recipe.b_recipe_bool_change THEN
			b_recipe_was_changed_bool:=TRUE;		
			IF gvl_recipe.s_recupe_change_4="false" THEN
				lr_old_param_bool:=0;
				lr_new_param_bool:=1;
			END_IF
			IF gvl_recipe.s_recupe_change_4="true" THEN
				lr_old_param_bool:=1;
				lr_new_param_bool:=0;
			END_IF
		//END_IF		
	END_IF
END_IF

IF b_recipe_bool_change.q OR b_recipe_real_change.q THEN
	FOR i := 499 TO 1 BY -1 DO
		gvl_recipe.ArRecipeChanges[i].old_value:=gvl_recipe.ArRecipeChanges[i-1].old_value;
		gvl_recipe.ArRecipeChanges[i].new_value:=gvl_recipe.ArRecipeChanges[i-1].new_value;
		gvl_recipe.ArRecipeChanges[i].when_changed:=gvl_recipe.ArRecipeChanges[i-1].when_changed;
		gvl_recipe.ArRecipeChanges[i].who_changed:=gvl_recipe.ArRecipeChanges[i-1].who_changed;
		gvl_recipe.ArRecipeChanges[i].which_param_name:=gvl_recipe.ArRecipeChanges[i-1].which_param_name;
		gvl_recipe.ArRecipeChanges[i].which_param_var:=gvl_recipe.ArRecipeChanges[i-1].which_param_var;
		gvl_recipe.ArRecipeChanges[i].which_param_cntr:=gvl_recipe.ArRecipeChanges[i-1].which_param_cntr;
		gvl_recipe.ArRecipeChanges[i].which_recipe:=gvl_recipe.ArRecipeChanges[i-1].which_recipe;
	END_FOR
END_IF
IF b_recipe_was_changed_real THEN
		gvl_recipe.ArRecipeChanges[0].old_value:=gvl_recipe.lr_recipe_change;
		gvl_recipe.ArRecipeChanges[0].new_value:=gvl_recipe.lr_recipe_change_1;
		gvl_recipe.ArRecipeChanges[0].when_changed:=P_time.actual_date_meawhile;
		gvl_recipe.ArRecipeChanges[0].who_changed:=gvl_recipe.s_recipe_change;
		gvl_recipe.ArRecipeChanges[0].which_param_name:=gvl_recipe.s_recipe_change_1;
		gvl_recipe.ArRecipeChanges[0].which_param_var:=wconcat(" '' ",gvl_recipe.s_recipe_change_2);
		gvl_recipe.ArRecipeChanges[0].which_param_cntr:=Wconcat("'",gvl_recipe.s_recipe_change_3);
		gvl_recipe.ArRecipeChanges[0].which_param_cntr:=Wconcat(gvl_recipe.ArRecipeChanges[0].which_param_cntr,"'");
		gvl_recipe.ArRecipeChanges[0].which_recipe:=gvl_recipe.s_recipe_name;
	END_IF
IF b_recipe_was_changed_bool THEN
		gvl_recipe.ArRecipeChanges[0].old_value:=lr_old_param_bool;
		gvl_recipe.ArRecipeChanges[0].new_value:=lr_new_param_bool;
		gvl_recipe.ArRecipeChanges[0].when_changed:=P_time.actual_date_meawhile;
		gvl_recipe.ArRecipeChanges[0].who_changed:=gvl_recipe.s_recipe_change;
		gvl_recipe.ArRecipeChanges[0].which_param_name:=gvl_recipe.s_recipe_change_1;
		gvl_recipe.ArRecipeChanges[0].which_param_var:=wconcat(" '' ",gvl_recipe.s_recipe_change_2);
		gvl_recipe.ArRecipeChanges[0].which_param_cntr:=Wconcat("'",gvl_recipe.s_recipe_change_3);
		gvl_recipe.ArRecipeChanges[0].which_param_cntr:=Wconcat(gvl_recipe.ArRecipeChanges[0].which_param_cntr,"'");
		gvl_recipe.ArRecipeChanges[0].which_recipe:=gvl_recipe.s_recipe_name;
END_IF

IF b_clear_recipe_history OR gvl_recipe.b_recipe_changes_clear THEN
	p_arraytofile.nFileCounter:=1;
FOR nIndex := 0 TO nTotalItems DO
    gvl_Recipe.ArRecipeChanges[nIndex].old_value := 0.0;
    gvl_Recipe.ArRecipeChanges[nIndex].new_value := 0.0;
    gvl_Recipe.ArRecipeChanges[nIndex].who_changed := "";         // WSTRING pusty
    gvl_Recipe.ArRecipeChanges[nIndex].when_changed := DT#1970-01-01-00:00:00; // Wartość domyślna dla DT
    gvl_Recipe.ArRecipeChanges[nIndex].which_param_name := "";     // WSTRING pusty
    gvl_Recipe.ArRecipeChanges[nIndex].which_param_var := "";      // WSTRING pusty
	gvl_recipe.ArRecipeChanges[nIndex].which_param_cntr:="";
	gvl_recipe.ArRecipeChanges[nIndex].which_recipe:="";
END_FOR
END_IF

IF gvl_recipe.ArRecipeChanges[400].which_param_cntr<>"" THEN
	b_clear_recipe_history:=TRUE;	
END_IF
		
IF gvl_recipe.b_recipe_bool_change=FALSE THEN
	b_recipe_was_changed_bool:=FALSE;
END_IF

IF gvl_recipe.b_recipe_real_change=FALSE THEN
		b_recipe_was_changed_real:=FALSE;
END_IF

END_PROGRAM

// ---- POUs/DataLogging/P_ArrayToFile.TcPOU
PROGRAM P_ArrayToFile
VAR
    fbFileOpen   : FB_FileOpen;
    fbFileClose  : FB_FileClose;
    fbFileWrite  : FB_FileWrite;
    hFile        : UINT := 0;(* File handle *)

    sFilePath    : STRING(400); //:= 'C:\Recipe_changes\RecipeChanges.txt'
    bSave        : BOOL;(* Trigger to start the file saving *)
    bBusy        : BOOL;
    bError       : BOOL;
    nErrId       : UDINT;
    
    Step         : DWORD := 0;(* Step for state machine *)
    nIndex       : INT := 0;(* Index for array iteration *)
    sBuffer      : STRING(255);(* Buff	er for writing to file *)
    nBytesToWrite: DINT;
    dtString     : STRING(25);
    nTotalItems  : INT := 500;(* Total items in array *)
	
    RisingEdge   : R_TRIG;


i:int;
	ColIndex: INT := 500;
	DataArray:ARRAY[0..500]OF INT;
END_VAR
VAR_INPUT
	nFileCounter :INT:=2;
END_VAR

RisingEdge(CLK := bSave OR gvl_recipe.b_recipe_bool_change OR gvl_recipe.b_recipe_real_change );

CASE Step OF
    0:
        IF RisingEdge.Q THEN
            bBusy := TRUE;
            bError := FALSE;
            nErrId := 0;
            nIndex := 0;
            Step := 10;
			sFilePath := CONCAT('C:\Recipe_changes\RecipeChanges_', INT_TO_STRING(nFileCounter));
			//sFilePath := CONCAT(sFilePath,dtString);
			sFilePath := CONCAT(sFilePath, '.txt'); 
			
			nFileCounter := nFileCounter + 1;
        END_IF

    10:
        fbFileOpen(sNetId := '', sPathName := sFilePath, 
                   nMode := FOPEN_MODEWRITE OR FOPEN_MODETEXT, 
                   ePath := PATH_GENERIC, 
                   bExecute := TRUE);      
		
			Step := 20;
		

		
    20:
        fbFileOpen(bExecute := FALSE);
        IF NOT fbFileOpen.bBusy THEN
            IF fbFileOpen.bError THEN
                nErrId := fbFileOpen.nErrId;
                bError := TRUE;
                Step := 500;
            ELSE
                hFile := fbFileOpen.hFile;
				i:=0;
                Step := 30;
            END_IF
        END_IF


    30:
        IF nIndex < nTotalItems THEN
            dtString := DT_TO_STRING(gvl_Recipe.ArRecipeChanges[nIndex].when_changed);
            sBuffer := CONCAT(CONCAT('Old Value: ', REAL_TO_STRING(gvl_Recipe.ArRecipeChanges[nIndex].old_value)), ' | ');
            sBuffer := CONCAT(sBuffer, CONCAT('New Value: ', REAL_TO_STRING(gvl_Recipe.ArRecipeChanges[nIndex].new_value)));
            sBuffer := CONCAT(sBuffer, CONCAT(' | Who Changed: ', WSTRING_TO_STRING(gvl_Recipe.ArRecipeChanges[nIndex].who_changed)));
            sBuffer := CONCAT(sBuffer, CONCAT(' | When Changed: ', dtString));
            sBuffer := CONCAT(sBuffer, CONCAT(' | Param Name: ', WSTRING_TO_STRING(gvl_Recipe.ArRecipeChanges[nIndex].which_param_name)));
            sBuffer := CONCAT(sBuffer, CONCAT(' | Param Var: ', WSTRING_TO_STRING(gvl_Recipe.ArRecipeChanges[nIndex].which_param_var)));
			sBuffer :=Concat(sBuffer, concat(' | Recipe name: ', WSTRING_TO_STRING(gvl_recipe.ArRecipeChanges[nIndex].which_recipe)));
            
		
			
			
			
			
            nBytesToWrite := LEN(sBuffer);
            
            fbFileWrite(sNetId := '', hFile := hFile, 
                        pWriteBuff := ADR(sBuffer), 
                        cbWriteLen := nBytesToWrite, 
                        bExecute := TRUE);
            Step := 40;
        ELSE
            Step := 300;
        END_IF

    40:
        fbFileWrite(bExecute := FALSE);
        IF NOT fbFileWrite.bBusy THEN
            IF fbFileWrite.bError THEN
                nErrId := fbFileWrite.nErrId;
                bError := TRUE;
                Step := 500;
            ELSE
                nIndex := nIndex + 1;
                Step := 30;
            END_IF
        END_IF

    300:
        fbFileClose(sNetId := '', hFile := hFile, bExecute := TRUE);
        Step := 310;

    310:
        fbFileClose(bExecute := FALSE);
        IF NOT fbFileClose.bBusy THEN
            IF fbFileClose.bError THEN
                nErrId := fbFileClose.nErrId;
                bError := TRUE;
            END_IF
            Step := 500;
        END_IF

    500:
        bBusy := FALSE;
        bSave := FALSE;
        Step := 0;
		ColIndex:=0;

END_CASE

END_PROGRAM

// ---- POUs/DataLogging/P_ScrewersCharts_1.TcPOU
PROGRAM P_ScrewersCharts_1


VAR
    fbFileOpen   : FB_FileOpen;
    fbFileClose  : FB_FileClose;
    fbFileWrite  : FB_FileWrite;
    hFile        : UINT := 0;(* File handle *)

    sFilePath    : STRING(400); //:= 'C:\Recipe_changes\RecipeChanges.txt'
    bSave        : BOOL;(* Trigger to start the file saving *)
    bBusy        : BOOL;
    bError       : BOOL;
    nErrId       : UDINT;
    
    Step         : DWORD := 0;(* Step for state machine *)
    nIndex       : INT := 0;(* Index for array iteration *)
    sBuffer      : STRING(3000);(* Buff	er for writing to file *)
    nBytesToWrite: DINT;
    dtString     : STRING(25);
    nTotalItems  : INT := 500;(* Total items in array *)
	nZeroCountInBuffer:int;
    RisingEdge   : R_TRIG;
	bNonZeroDetected:BOOL;
	nZeroCount:INT;
	i:INT;
	nDataLength:INT;
	ColIndex: INT := 500;
	DataArray:ARRAY[0..500]OF INT;
	ftbRun:f_trig;
	
    nIndex_l: INT := 1;
    bWrite1: BOOL; 
	bWrite2: BOOL;
    nValueToWrite: INT; 
    bError1: BOOL := FALSE;
    nErrId1: UINT; 
	bhandy1:bool;
	
	lrPreviousValueTorqueSetted:LREAL;
	
	
	
	
END_VAR
VAR_INPUT
	nFileCounter :INT:=2;
END_VAR


//P10_GripperScrewer.fb2GripperScrewer1.bCycleDone1

ftbRun(clk:= P_ADS_SCREW.bScrewer1Run);
RisingEdge(CLK := ftbRun.Q );//OR P_ADS_Screw.bScrewer1Done1 OR P_ADS_Screw.bScrewer1Done2 OR P_ADS_Screw.bScrewer1NotDone1 OR ftbRun.q);
CASE Step OF
    0:
        IF RisingEdge.Q THEN
            bBusy := TRUE;
            bError := FALSE;
            nErrId := 0;
            nIndex := 0;
            sFilePath := CONCAT('C:\LastScrewingCycles\Zakrecarka_1_', INT_TO_STRING(nFileCounter));
            sFilePath := CONCAT(sFilePath, '.csv');
            nFileCounter := nFileCounter + 1;
            IF nFileCounter > 50 THEN
                nFileCounter := 1;
            END_IF
            Step := 10;
        END_IF
    10:
        // Kopiowanie wszystkich danych do DataArray
        FOR i := 0 TO 500 DO
            DataArray[i] := P_ADS_Screw.AStChartGripperScrewer1[0][2, i];
        END_FOR
        nDataLength := 500; // Ustaw pełną długość danych
        Step := 20;
    20:
        // Otwórz plik do zapisu
        fbFileOpen(sNetId := '', sPathName := sFilePath,
                   nMode := FOPEN_MODEWRITE OR FOPEN_MODETEXT,
                   ePath := PATH_GENERIC,
                   bExecute := TRUE);
        Step := 30;
    30:
        fbFileOpen(bExecute := FALSE);
        IF NOT fbFileOpen.bBusy THEN
            IF fbFileOpen.bError THEN
                nErrId := fbFileOpen.nErrId;
                bError := TRUE;
                Step := 500;
            ELSE
                hFile := fbFileOpen.hFile;
                Step := 40;
            END_IF
        END_IF
    40:
        // Zapisz dane w mniejszych porcjach (np. po 100 wierszy)
        IF nIndex <= nDataLength THEN
            sBuffer := '';
            FOR i := nIndex TO MIN(nIndex + 99, nDataLength) DO
                sBuffer := CONCAT(sBuffer, INT_TO_STRING(DataArray[i]));
				sBuffer := CONCAT(sBuffer, '$N');
            END_FOR
            nBytesToWrite := LEN(sBuffer);
            fbFileWrite(sNetId := '', hFile := hFile,
                        pWriteBuff := ADR(sBuffer),
                        cbWriteLen := nBytesToWrite,
                        bExecute := TRUE);
            Step := 50;
        ELSE
            Step := 300; // Przejdź do zamknięcia pliku po zapisaniu wszystkich danych
        END_IF
    50:
        fbFileWrite(bExecute := FALSE);
        IF NOT fbFileWrite.bBusy THEN
            IF fbFileWrite.bError THEN
                nErrId := fbFileWrite.nErrId;
                bError := TRUE;
                Step := 500;
            ELSE
                nIndex := nIndex + 100; // Przejdź do następnej porcji danych
                Step := 40;
            END_IF
        END_IF
    300:
        // Zamknij plik
        fbFileClose(sNetId := '', hFile := hFile, bExecute := TRUE);
        Step := 310;
    310:
        fbFileClose(bExecute := FALSE);
        IF NOT fbFileClose.bBusy THEN
            IF fbFileClose.bError THEN
                nErrId := fbFileClose.nErrId;
                bError := TRUE;
            END_IF
            Step := 500;
        END_IF
    500:
        // Zakończ eksport
        bBusy := FALSE;
        bSave := FALSE;
        Step := 0;
        nIndex := 0; 
END_CASE

bWrite1:=ftbRun.q;
IF bWrite1 THEN
    IF nValueToWrite >= 0 THEN
        gvl_screw.aLast50Screw1[nIndex_l] := p_ads_screw.lrGripperScrewer1TorqueCV;
        nIndex_l := nIndex_l + 1;
        IF nIndex_l > 500 THEN
            nIndex_l := 1;
        END_IF;
        bWrite1 := FALSE;
    ELSE
        bError1 := TRUE;
        nErrId1 := 1;
    END_IF;
END_IF;

IF lrPreviousValueTorqueSetted<>P_ADS_SCREW.lrGripperScrewingTightTorqueShow OR bhandy1 THEN
	for i:=1 to 501 do
		gvl_screw.a50ScrewSetted1[i]:=P_ADS_SCREW.lrGripperScrewingTightTorqueShow;
	END_FOR
	lrPreviousValueTorqueSetted:=P_ADS_SCREW.lrGripperScrewingTightTorqueShow;
END_IF;

END_PROGRAM

// ---- POUs/ADS/P_ADS_Screw.TcPOU
PROGRAM P_ADS_Screw
VAR
	bTrigger				: BOOL;
		
//pliki zakręcarek
	fbRead_19:	FB_ReadAdsSymByName;
	AStChartGripperScrewer1	:ARRAY[0..100] OF ARRAY[0..5, 0..500] OF INT;
	fbCyclicReadout: TON;
	
	fbRead_20:	FB_ReadAdsSymByName;
	bScrewer1Done1 :BOOL;
	bScrewer1Done2 :BOOL;
	fbRead_21:	FB_ReadAdsSymByName;
	bScrewer2Done1 :BOOL;
	bScrewer2Done2 :BOOL;
	fbRead_22:	FB_ReadAdsSymByName;
	fbRead_23:	FB_ReadAdsSymByName;
	fbRead_24:	FB_ReadAdsSymByName;
	fbRead_25:	FB_ReadAdsSymByName;
	fbRead_26:	FB_ReadAdsSymByName;
	AStChartGripperScrewer2	:ARRAY[0..100] OF ARRAY[0..5, 0..500] OF INT;
	bScrewer1NotDone1 :BOOL;
	bScrewer2NotDone1 :BOOL;
	bScrewer1Run:BOOL;
	bScrewer2Run:BOOL;
	fbRead_27:	FB_ReadAdsSymByName;
	fbRead_28:	FB_ReadAdsSymByName;
	fbRead_29:	FB_ReadAdsSymByName;
	fbRead_30:	FB_ReadAdsSymByName;	
	lrGripperScrewer1TorqueCV :LREAL;
	lrGripperScrewer2TorqueCV :LREAL;
	fbRead_31:	FB_ReadAdsSymByName;
	fbRead_32:	FB_ReadAdsSymByName;
	lrGripperScrewingTightTorqueShow:LREAL;
	lrGripperScrewing2TightTorqueShow:LREAL;
END_VAR

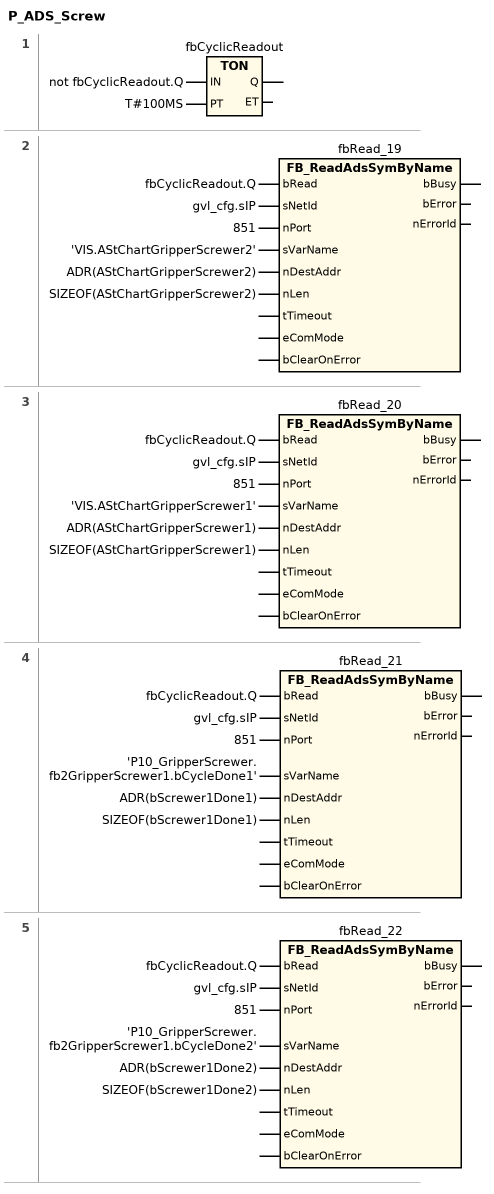
// NETWORK 1
fbCyclicReadout(IN := not fbCyclicReadout.Q, PT := T#100MS); // TON

// NETWORK 2
fbRead_19(
    bRead := fbCyclicReadout.Q,
    sNetId := gvl_cfg.sIP,
    nPort := 851,
    sVarName := 'VIS.AStChartGripperScrewer2',
    nDestAddr := ADR(AStChartGripperScrewer2),
    nLen := SIZEOF(AStChartGripperScrewer2)); // FB_ReadAdsSymByName

// NETWORK 3
fbRead_20(
    bRead := fbCyclicReadout.Q,
    sNetId := gvl_cfg.sIP,
    nPort := 851,
    sVarName := 'VIS.AStChartGripperScrewer1',
    nDestAddr := ADR(AStChartGripperScrewer1),
    nLen := SIZEOF(AStChartGripperScrewer1)); // FB_ReadAdsSymByName

// NETWORK 4
fbRead_21(
    bRead := fbCyclicReadout.Q,
    sNetId := gvl_cfg.sIP,
    nPort := 851,
    sVarName := 'P10_GripperScrewer.fb2GripperScrewer1.bCycleDone1',
    nDestAddr := ADR(bScrewer1Done1),
    nLen := SIZEOF(bScrewer1Done1)); // FB_ReadAdsSymByName

// NETWORK 5
fbRead_22(
    bRead := fbCyclicReadout.Q,
    sNetId := gvl_cfg.sIP,
    nPort := 851,
    sVarName := 'P10_GripperScrewer.fb2GripperScrewer1.bCycleDone2',
    nDestAddr := ADR(bScrewer1Done2),
    nLen := SIZEOF(bScrewer1Done2)); // FB_ReadAdsSymByName

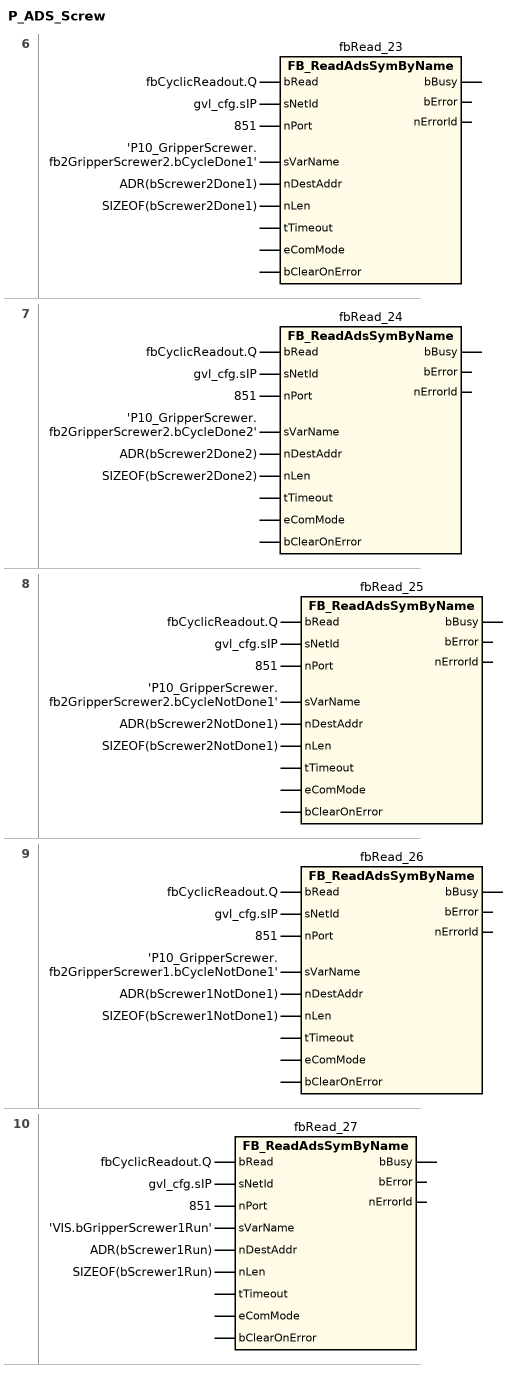
// NETWORK 6
fbRead_23(
    bRead := fbCyclicReadout.Q,
    sNetId := gvl_cfg.sIP,
    nPort := 851,
    sVarName := 'P10_GripperScrewer.fb2GripperScrewer2.bCycleDone1',
    nDestAddr := ADR(bScrewer2Done1),
    nLen := SIZEOF(bScrewer2Done1)); // FB_ReadAdsSymByName

// NETWORK 7
fbRead_24(
    bRead := fbCyclicReadout.Q,
    sNetId := gvl_cfg.sIP,
    nPort := 851,
    sVarName := 'P10_GripperScrewer.fb2GripperScrewer2.bCycleDone2',
    nDestAddr := ADR(bScrewer2Done2),
    nLen := SIZEOF(bScrewer2Done2)); // FB_ReadAdsSymByName

// NETWORK 8
fbRead_25(
    bRead := fbCyclicReadout.Q,
    sNetId := gvl_cfg.sIP,
    nPort := 851,
    sVarName := 'P10_GripperScrewer.fb2GripperScrewer2.bCycleNotDone1',
    nDestAddr := ADR(bScrewer2NotDone1),
    nLen := SIZEOF(bScrewer2NotDone1)); // FB_ReadAdsSymByName

// NETWORK 9
fbRead_26(
    bRead := fbCyclicReadout.Q,
    sNetId := gvl_cfg.sIP,
    nPort := 851,
    sVarName := 'P10_GripperScrewer.fb2GripperScrewer1.bCycleNotDone1',
    nDestAddr := ADR(bScrewer1NotDone1),
    nLen := SIZEOF(bScrewer1NotDone1)); // FB_ReadAdsSymByName

// NETWORK 10
fbRead_27(
    bRead := fbCyclicReadout.Q,
    sNetId := gvl_cfg.sIP,
    nPort := 851,
    sVarName := 'VIS.bGripperScrewer1Run',
    nDestAddr := ADR(bScrewer1Run),
    nLen := SIZEOF(bScrewer1Run)); // FB_ReadAdsSymByName

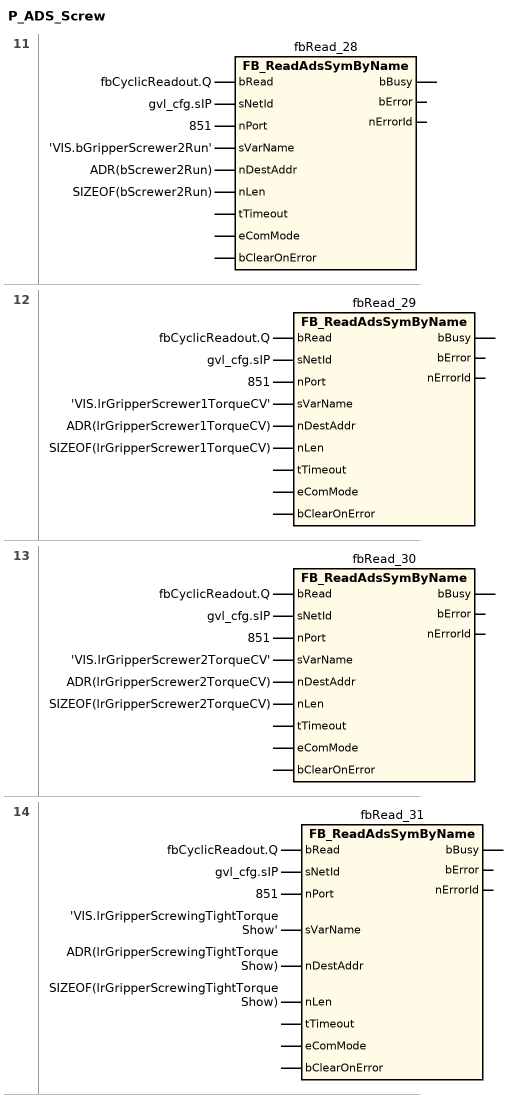
// NETWORK 11
fbRead_28(
    bRead := fbCyclicReadout.Q,
    sNetId := gvl_cfg.sIP,
    nPort := 851,
    sVarName := 'VIS.bGripperScrewer2Run',
    nDestAddr := ADR(bScrewer2Run),
    nLen := SIZEOF(bScrewer2Run)); // FB_ReadAdsSymByName

// NETWORK 12
fbRead_29(
    bRead := fbCyclicReadout.Q,
    sNetId := gvl_cfg.sIP,
    nPort := 851,
    sVarName := 'VIS.lrGripperScrewer1TorqueCV',
    nDestAddr := ADR(lrGripperScrewer1TorqueCV),
    nLen := SIZEOF(lrGripperScrewer1TorqueCV)); // FB_ReadAdsSymByName

// NETWORK 13
fbRead_30(
    bRead := fbCyclicReadout.Q,
    sNetId := gvl_cfg.sIP,
    nPort := 851,
    sVarName := 'VIS.lrGripperScrewer2TorqueCV',
    nDestAddr := ADR(lrGripperScrewer2TorqueCV),
    nLen := SIZEOF(lrGripperScrewer2TorqueCV)); // FB_ReadAdsSymByName

// NETWORK 14
fbRead_31(
    bRead := fbCyclicReadout.Q,
    sNetId := gvl_cfg.sIP,
    nPort := 851,
    sVarName := 'VIS.lrGripperScrewingTightTorqueShow',
    nDestAddr := ADR(lrGripperScrewingTightTorqueShow),
    nLen := SIZEOF(lrGripperScrewingTightTorqueShow)); // FB_ReadAdsSymByName

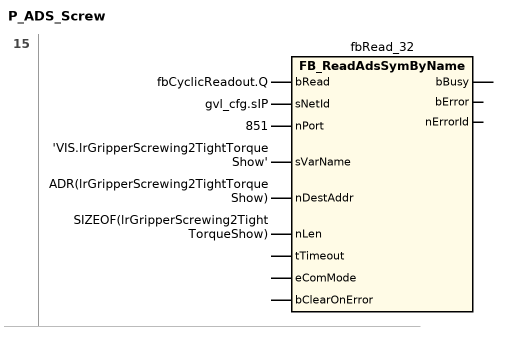
// NETWORK 15
fbRead_32(
    bRead := fbCyclicReadout.Q,
    sNetId := gvl_cfg.sIP,
    nPort := 851,
    sVarName := 'VIS.lrGripperScrewing2TightTorqueShow',
    nDestAddr := ADR(lrGripperScrewing2TightTorqueShow),
    nLen := SIZEOF(lrGripperScrewing2TightTorqueShow)); // FB_ReadAdsSymByName

END_PROGRAM

// ---- POUs/DataLogging/P_ScrewersCharts_2.TcPOU
PROGRAM P_ScrewersCharts_2


VAR
    fbFileOpen   : FB_FileOpen;
    fbFileClose  : FB_FileClose;
    fbFileWrite  : FB_FileWrite;
    hFile        : UINT := 0;(* File handle *)

    sFilePath    : STRING(400); //:= 'C:\Recipe_changes\RecipeChanges.txt'
    bSave        : BOOL;(* Trigger to start the file saving *)
    bBusy        : BOOL;
    bError       : BOOL;
    nErrId       : UDINT;
    
    Step         : DWORD := 0;(* Step for state machine *)
    nIndex       : INT := 0;(* Index for array iteration *)
    sBuffer      : STRING(255);(* Buff	er for writing to file *)
    nBytesToWrite: DINT;
    dtString     : STRING(25);
    nTotalItems  : INT := 500;(* Total items in array *)
	nZeroCountInBuffer:INT;
    RisingEdge   : R_TRIG;
	nDataLength:INT;
	bNonZeroDetected:BOOL;
	i:INT;
	nZeroCount:INT;
	ftbRun:F_trig;
	ColIndex: INT := 500;
	DataArray:ARRAY[0..500]OF INT;
	  nIndex_l: INT := 1;
    bWrite1: BOOL; 
	bWrite2: BOOL;
    nValueToWrite: INT; 
    bError1: BOOL := FALSE;
    nErrId1: UINT; 
	bhandy1:bool;
	lrPreviousValueTorqueSetted: LREAL;
END_VAR
VAR_INPUT
	nFileCounter :INT:=2;
END_VAR


//P10_GripperScrewer.fb2GripperScrewer1.bCycleDone1

ftbRun(clk:= P_ADS_SCREW.bScrewer2Run);
RisingEdge(clk:=ftbrun.Q); //CLK := bSave OR P_ADS_Screw.bScrewer2Done1 OR P_ADS_Screw.bScrewer2Done2 OR P_ADS_Screw.bScrewer2NotDone1 OR ftbrun.Q);
CASE Step OF
    0:
        IF RisingEdge.Q THEN
            bBusy := TRUE;
            bError := FALSE;
            nErrId := 0;
            nIndex := 0;
            sFilePath := CONCAT('C:\LastScrewingCycles\Zakrecarka_2_', INT_TO_STRING(nFileCounter));
            sFilePath := CONCAT(sFilePath, '.csv');
            nFileCounter := nFileCounter + 1;
            IF nFileCounter > 50 THEN
                nFileCounter := 1;
            END_IF
            Step := 10;
        END_IF
    10:

        FOR i := 0 TO 500 DO
            DataArray[i] := P_ADS_Screw.AStChartGripperScrewer2[0][2, i];
        END_FOR
        nDataLength := 500;
        Step := 20;
    20:
      
        fbFileOpen(sNetId := '', sPathName := sFilePath,
                   nMode := FOPEN_MODEWRITE OR FOPEN_MODETEXT,
                   ePath := PATH_GENERIC,
                   bExecute := TRUE);
        Step := 30;
    30:
        fbFileOpen(bExecute := FALSE);
        IF NOT fbFileOpen.bBusy THEN
            IF fbFileOpen.bError THEN
                nErrId := fbFileOpen.nErrId;
                bError := TRUE;
                Step := 500;
            ELSE
                hFile := fbFileOpen.hFile;
                Step := 40;
            END_IF
        END_IF
    40:
       
        IF nIndex <= nDataLength THEN
            sBuffer := '';
            FOR i := nIndex TO MIN(nIndex + 99, nDataLength) DO
                sBuffer := CONCAT(sBuffer, INT_TO_STRING(DataArray[i]));
				sBuffer := CONCAT(sBuffer, '$N');
            END_FOR
            nBytesToWrite := LEN(sBuffer);
            fbFileWrite(sNetId := '', hFile := hFile,
                        pWriteBuff := ADR(sBuffer),
                        cbWriteLen := nBytesToWrite,
                        bExecute := TRUE);
            Step := 50;
        ELSE
            Step := 300; 
        END_IF
    50:
        fbFileWrite(bExecute := FALSE);
        IF NOT fbFileWrite.bBusy THEN
            IF fbFileWrite.bError THEN
                nErrId := fbFileWrite.nErrId;
                bError := TRUE;
                Step := 500;
            ELSE
                nIndex := nIndex + 100;
                Step := 40;
            END_IF
        END_IF
    300:
       
        fbFileClose(sNetId := '', hFile := hFile, bExecute := TRUE);
        Step := 310;
    310:
        fbFileClose(bExecute := FALSE);
        IF NOT fbFileClose.bBusy THEN
            IF fbFileClose.bError THEN
                nErrId := fbFileClose.nErrId;
                bError := TRUE;
            END_IF
            Step := 500;
        END_IF
    500:
     
        bBusy := FALSE;
        bSave := FALSE;
        Step := 0;
        nIndex := 0;
END_CASE



bWrite1:=ftbRun.q;
IF bWrite1 THEN
    IF nValueToWrite >= 0 THEN
        gvl_screw.aLast50Screw2[nIndex_l] := p_ads_screw.lrGripperScrewer2TorqueCV;
        nIndex_l := nIndex_l + 1;
        IF nIndex_l > 500 THEN
            nIndex_l := 1;
        END_IF;
        bWrite1 := FALSE;
    ELSE
        bError1 := TRUE;
        nErrId1 := 1;
    END_IF;
END_IF;


IF lrPreviousValueTorqueSetted<>P_ADS_SCREW.lrGripperScrewing2TightTorqueShow OR bhandy1 THEN
	FOR i:=1 TO 501 DO
		gvl_screw.a50ScrewSetted2[i]:=P_ADS_SCREW.lrGripperScrewing2TightTorqueShow;
	END_FOR
	lrPreviousValueTorqueSetted:=P_ADS_SCREW.lrGripperScrewing2TightTorqueShow;
END_IF;

END_PROGRAM

// ---- POUs/DataLogging/p_24h_C1_2.TcPOU
PROGRAM P_24h_C1_2
// Zmienne pomocnicze
VAR
    sCurrentDate        : STRING(10) := '';  // Przechowuje aktualną datę (np. "2023-10-25")
    bNewDay             : BOOL := FALSE;     // Flaga wskazująca, że rozpoczął się nowy dzień
    hFile               : UINT := 0;        // Uchwyt pliku
    sFilePath           : T_MaxString := ''; // Ścieżka do pliku
    nBytesToWrite       : UDINT := 0;        // Liczba bajtów do zapisania
    sLineToWrite             : T_MaxString := ''; // Bufor na dane do zapisania
    dtString            : STRING(20) := '';  // Czas zmiany w formacie tekstowym
    fbFileSeek          : FB_FileSeek;       // Blok do pozycjonowania wskaźnika pliku
    fbFileTell          : FB_FileTell;       // Blok do odczytu pozycji wskaźnika pliku
    fbFileGets          : FB_FileGets;       // Blok do odczytu linii z pliku
    bFileIsEmpty        : BOOL := FALSE;     // Flaga wskazująca, czy plik jest pusty
	RisingEdge			:R_trig;
	bSaveManuel			:BOOL;
	Step				:INT;
	bBusy 				:BOOL;
	bError				:BOOL;
	nErrId				:UDINT;
	nIndex				:INT;
	sFolderPath: STRING(255) := 'C:\Last24ScrewingCycles\';
	fbFileOpen: FB_FileOpen;
    fbFileWrite: FB_FileWrite;
    fbFileClose: FB_FileClose;
	b10step:BOOL;
	ftrig:F_trig;
END_VAR

// Główna logika
ftrig(CLK:=P_ADS_SCREW.bScrewer2Run);
RisingEdge(CLK := bSaveManuel OR ftrig.Q);

CASE Step OF
    0:
        // Sprawdź, czy zmienił się dzień
        IF LEFT(WSTRING_TO_STRING(P_time.s_time_mainscreen), 10) <> sCurrentDate THEN
            sCurrentDate := LEFT(WSTRING_TO_STRING(P_time.s_time_mainscreen), 10);  // Zaktualizuj datę
            bNewDay := TRUE;  // Ustaw flagę nowego dnia
        END_IF

        // Jeśli wystąpiło zdarzenie zapisu lub zmiany receptury
        IF RisingEdge.Q THEN
            bBusy := TRUE;
            bError := FALSE;
            nErrId := 0;
            nIndex := 0;

            // Utwórz ścieżkę do pliku na podstawie aktualnej daty
            sFilePath := CONCAT(sFolderPath, 'Capper_1_');
            sFilePath := CONCAT(sFilePath, sCurrentDate);
            sFilePath := CONCAT(sFilePath, '.csv');

            Step := 10;  // Przejdź do kroku otwarcia pliku
        END_IF

    10:
        // Otwórz plik
        IF bNewDay THEN
            // Jeśli nowy dzień, otwórz plik w trybie zapisu (tworzy nowy plik)
            fbFileOpen(
                sNetId := '', 
                sPathName := sFilePath, 
                nMode := FOPEN_MODEWRITE OR FOPEN_MODETEXT, 
                ePath := PATH_GENERIC, 
                bExecute := TRUE
            );
            b10step := TRUE;
        ELSE
            // Jeśli stary dzień, otwórz plik w trybie dopisywania
            fbFileOpen(
                sNetId := '', 
                sPathName := sFilePath, 
                nMode := FOPEN_MODEAPPEND OR FOPEN_MODETEXT, 
                ePath := PATH_GENERIC, 
                bExecute := TRUE
            );
            b10step := TRUE;
        END_IF
        Step := 20;

    20:
        // Czekaj na otwarcie pliku
        fbFileOpen(bExecute := FALSE);
        IF NOT fbFileOpen.bBusy THEN
            IF fbFileOpen.bError THEN
                nErrId := fbFileOpen.nErrId;
                bError := TRUE;
                Step := 500;  // Przejdź do kroku obsługi błędów
            ELSE
                hFile := fbFileOpen.hFile;
                Step := 30;  // Przejdź do kroku weryfikacji pliku
            END_IF
        END_IF

    30:
        // Sprawdź, czy plik jest pusty (tylko dla nowego dnia)
        IF bNewDay THEN
            fbFileTell(
                sNetId := '', 
                hFile := hFile, 
                bExecute := TRUE
            );
            Step := 35;
        ELSE
            Step := 40;  // Pomijaj weryfikację dla starego dnia
        END_IF

    35:
        // Czekaj na odczyt pozycji wskaźnika pliku
        fbFileTell(bExecute := FALSE);
        IF NOT fbFileTell.bBusy THEN
            IF fbFileTell.nSeekPos = 0 THEN
                bFileIsEmpty := TRUE;  // Plik jest pusty
            ELSE
                bFileIsEmpty := FALSE; // Plik nie jest pusty
            END_IF
            Step := 40;
        END_IF

    40:
        // Przygotuj dane do zapisu
        IF NOT fbFileTell.bBusy THEN
            sLineToWrite := CONCAT(WSTRING_TO_STRING(P_time.s_time_mainscreen), ',');
            sLineToWrite := CONCAT(sLineToWrite, REAL_TO_STRING(P_ADS_SCREW.lrGripperScrewer1TorqueCV));
            sLineToWrite := CONCAT(sLineToWrite, ',');
            sLineToWrite := CONCAT(sLineToWrite, WSTRING_TO_STRING(gvl_recipe.s_recipe_name));
            sLineToWrite := CONCAT(sLineToWrite, '$N');

            nBytesToWrite := LEN(sLineToWrite);

            // Zapisz dane do pliku
            fbFileWrite(
                sNetId := '', 
                hFile := hFile, 
                pWriteBuff := ADR(sLineToWrite), 
                cbWriteLen := nBytesToWrite, 
                bExecute := TRUE
            );
            Step := 50;
        ELSE
            Step := 300;  // Przejdź do kroku zamknięcia pliku
        END_IF

    50:
        // Czekaj na zakończenie zapisu
        fbFileWrite(bExecute := FALSE);
        IF NOT fbFileWrite.bBusy THEN
            IF fbFileWrite.bError THEN
                nErrId := fbFileWrite.nErrId;
                bError := TRUE;
                Step := 500;  // Przejdź do kroku obsługi błędów
            ELSE
                Step := 300;  // Przejdź do kroku zamknięcia pliku po jednokrotnym zapisie
            END_IF
        END_IF

    300:
        // Zamknij plik
        fbFileClose(
            sNetId := '', 
            hFile := hFile, 
            bExecute := TRUE
        );
        Step := 310;

    310:
        // Czekaj na zamknięcie pliku
        fbFileClose(bExecute := FALSE);
        IF NOT fbFileClose.bBusy THEN
            IF fbFileClose.bError THEN
                nErrId := fbFileClose.nErrId;
                bError := TRUE;
            END_IF
            Step := 500;  // Przejdź do kroku obsługi błędów
        END_IF

    500:
        // Zakończ procedurę
        bBusy := FALSE;
        bNewDay := FALSE;  // Zresetuj flagę nowego dnia
        Step := 0;
END_CASE

END_PROGRAM

// ---- POUs/DataLogging/p_24h_C2_2.TcPOU
PROGRAM p_24h_C2_2
// Zmienne pomocnicze
VAR
    sCurrentDate        : STRING(10) := '';  // Przechowuje aktualną datę (np. "2023-10-25")
    bNewDay             : BOOL := FALSE;     // Flaga wskazująca, że rozpoczął się nowy dzień
    hFile               : UINT := 0;        // Uchwyt pliku
    sFilePath           : T_MaxString := ''; // Ścieżka do pliku
    nBytesToWrite       : UDINT := 0;        // Liczba bajtów do zapisania
    sLineToWrite             : T_MaxString := ''; // Bufor na dane do zapisania
    dtString            : STRING(20) := '';  // Czas zmiany w formacie tekstowym
    fbFileSeek          : FB_FileSeek;       // Blok do pozycjonowania wskaźnika pliku
    fbFileTell          : FB_FileTell;       // Blok do odczytu pozycji wskaźnika pliku
    fbFileGets          : FB_FileGets;       // Blok do odczytu linii z pliku
    bFileIsEmpty        : BOOL := FALSE;     // Flaga wskazująca, czy plik jest pusty
	RisingEdge			:R_trig;
	bSaveManuel			:BOOL;
	Step				:INT;
	bBusy 				:BOOL;
	bError				:BOOL;
	nErrId				:UDINT;
	nIndex				:INT;
	sFolderPath: STRING(255) := 'C:\Last24ScrewingCycles\';
	fbFileOpen: FB_FileOpen;
    fbFileWrite: FB_FileWrite;
    fbFileClose: FB_FileClose;
	b10step:BOOL;
	ftrig:F_trig;
END_VAR

// Główna logika
ftrig(CLK:=P_ADS_SCREW.bScrewer2Run);
RisingEdge(CLK := bSaveManuel OR ftrig.Q);

CASE Step OF
    0:
        // Sprawdź, czy zmienił się dzień
        IF LEFT(WSTRING_TO_STRING(P_time.s_time_mainscreen), 10) <> sCurrentDate THEN
            sCurrentDate := LEFT(WSTRING_TO_STRING(P_time.s_time_mainscreen), 10);  // Zaktualizuj datę
            bNewDay := TRUE;  // Ustaw flagę nowego dnia
        END_IF

        // Jeśli wystąpiło zdarzenie zapisu lub zmiany receptury
        IF RisingEdge.Q THEN
            bBusy := TRUE;
            bError := FALSE;
            nErrId := 0;
            nIndex := 0;

            // Utwórz ścieżkę do pliku na podstawie aktualnej daty
            sFilePath := CONCAT(sFolderPath, 'Capper_2_');
            sFilePath := CONCAT(sFilePath, sCurrentDate);
            sFilePath := CONCAT(sFilePath, '.csv');

            Step := 10;  // Przejdź do kroku otwarcia pliku
        END_IF

    10:
        // Otwórz plik
        IF bNewDay THEN
            // Jeśli nowy dzień, otwórz plik w trybie zapisu (tworzy nowy plik)
            fbFileOpen(
                sNetId := '', 
                sPathName := sFilePath, 
                nMode := FOPEN_MODEWRITE OR FOPEN_MODETEXT, 
                ePath := PATH_GENERIC, 
                bExecute := TRUE
            );
            b10step := TRUE;
        ELSE
            // Jeśli stary dzień, otwórz plik w trybie dopisywania
            fbFileOpen(
                sNetId := '', 
                sPathName := sFilePath, 
                nMode := FOPEN_MODEAPPEND OR FOPEN_MODETEXT, 
                ePath := PATH_GENERIC, 
                bExecute := TRUE
            );
            b10step := TRUE;
        END_IF
        Step := 20;

    20:
        // Czekaj na otwarcie pliku
        fbFileOpen(bExecute := FALSE);
        IF NOT fbFileOpen.bBusy THEN
            IF fbFileOpen.bError THEN
                nErrId := fbFileOpen.nErrId;
                bError := TRUE;
                Step := 500;  // Przejdź do kroku obsługi błędów
            ELSE
                hFile := fbFileOpen.hFile;
                Step := 30;  // Przejdź do kroku weryfikacji pliku
            END_IF
        END_IF

    30:
        // Sprawdź, czy plik jest pusty (tylko dla nowego dnia)
        IF bNewDay THEN
            fbFileTell(
                sNetId := '', 
                hFile := hFile, 
                bExecute := TRUE
            );
            Step := 35;
        ELSE
            Step := 40;  // Pomijaj weryfikację dla starego dnia
        END_IF

    35:
        // Czekaj na odczyt pozycji wskaźnika pliku
        fbFileTell(bExecute := FALSE);
        IF NOT fbFileTell.bBusy THEN
            IF fbFileTell.nSeekPos = 0 THEN
                bFileIsEmpty := TRUE;  // Plik jest pusty
            ELSE
                bFileIsEmpty := FALSE; // Plik nie jest pusty
            END_IF
            Step := 40;
        END_IF

    40:
        // Przygotuj dane do zapisu
        IF NOT fbFileTell.bBusy THEN
            sLineToWrite := CONCAT(WSTRING_TO_STRING(P_time.s_time_mainscreen), ',');
            sLineToWrite := CONCAT(sLineToWrite, REAL_TO_STRING(P_ADS_SCREW.lrGripperScrewer2TorqueCV));
            sLineToWrite := CONCAT(sLineToWrite, ',');
            sLineToWrite := CONCAT(sLineToWrite, WSTRING_TO_STRING(gvl_recipe.s_recipe_name));
            sLineToWrite := CONCAT(sLineToWrite, '$N');

            nBytesToWrite := LEN(sLineToWrite);

            // Zapisz dane do pliku
            fbFileWrite(
                sNetId := '', 
                hFile := hFile, 
                pWriteBuff := ADR(sLineToWrite), 
                cbWriteLen := nBytesToWrite, 
                bExecute := TRUE
            );
            Step := 50;
        ELSE
            Step := 300;  // Przejdź do kroku zamknięcia pliku
        END_IF

    50:
        // Czekaj na zakończenie zapisu
        fbFileWrite(bExecute := FALSE);
        IF NOT fbFileWrite.bBusy THEN
            IF fbFileWrite.bError THEN
                nErrId := fbFileWrite.nErrId;
                bError := TRUE;
                Step := 500;  // Przejdź do kroku obsługi błędów
            ELSE
                Step := 300;  // Przejdź do kroku zamknięcia pliku po jednokrotnym zapisie
            END_IF
        END_IF

    300:
        // Zamknij plik
        fbFileClose(
            sNetId := '', 
            hFile := hFile, 
            bExecute := TRUE
        );
        Step := 310;

    310:
        // Czekaj na zamknięcie pliku
        fbFileClose(bExecute := FALSE);
        IF NOT fbFileClose.bBusy THEN
            IF fbFileClose.bError THEN
                nErrId := fbFileClose.nErrId;
                bError := TRUE;
            END_IF
            Step := 500;  // Przejdź do kroku obsługi błędów
        END_IF

    500:
        // Zakończ procedurę
        bBusy := FALSE;
        bNewDay := FALSE;  // Zresetuj flagę nowego dnia
        Step := 0;
END_CASE

END_PROGRAM

// ---- POUs/DataLogging/P_CameraFlip.TcPOU
PROGRAM P_CameraFlip
VAR
	fbFileOpen: FB_FileOpen;
    fbFileWrite: FB_FileWrite;
    fbFileClose: FB_FileClose;
    hFile : UINT;
    nResultCreate, nResultDelete : INT;
    sPath : STRING := 'C:\Users\Administrator\Desktop\CameraFlip\trigger.txt';
    bFileExists : BOOL;
	Step:INT;
	ftrig:F_trig;
	RisingEdge:R_trig;
	bBusy 				:BOOL;
	bError				:BOOL;
	nErrId				:UDINT;
    nIndex				:INT;
END_VAR

RisingEdge(CLK := gvl_error.b_cameras_ivms);

CASE Step OF
    0:
        // Jeśli wystąpiło zdarzenie zapisu lub zmiany receptury
        IF RisingEdge.Q THEN
            bBusy := TRUE;
            bError := FALSE;
            nErrId := 0;
            nIndex := 0;

